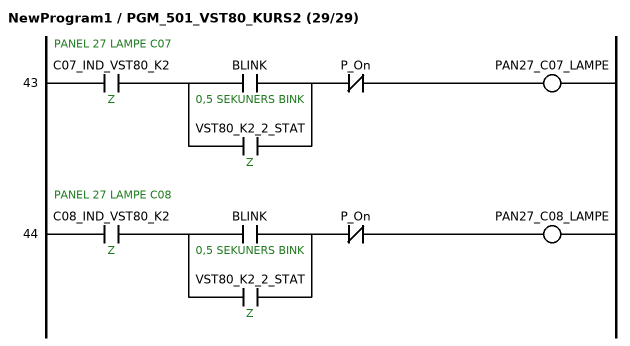
; [picture p528: NewProgram1 / PGM_501_VST80_KURS2, rungs 43-44]
; rung 43: PANEL 27 LAMPE C07
LD C07_IND_VST80_K2  ; Z
LD BLINK  ; 0,5 SEKUNERS BINK
OR VST80_K2_2_STAT  ; Z
ANDLD
ANDNOT P_On
OUT PAN27_C07_LAMPE
; rung 44: PANEL 27 LAMPE C08
LD C08_IND_VST80_K2  ; Z
LD BLINK  ; 0,5 SEKUNERS BINK
OR VST80_K2_2_STAT  ; Z
ANDLD
ANDNOT P_On
OUT PAN27_C08_LAMPE
; rung 45: Ingen_kommentar_funnet

### Section PGM_502_VST80_KURS3

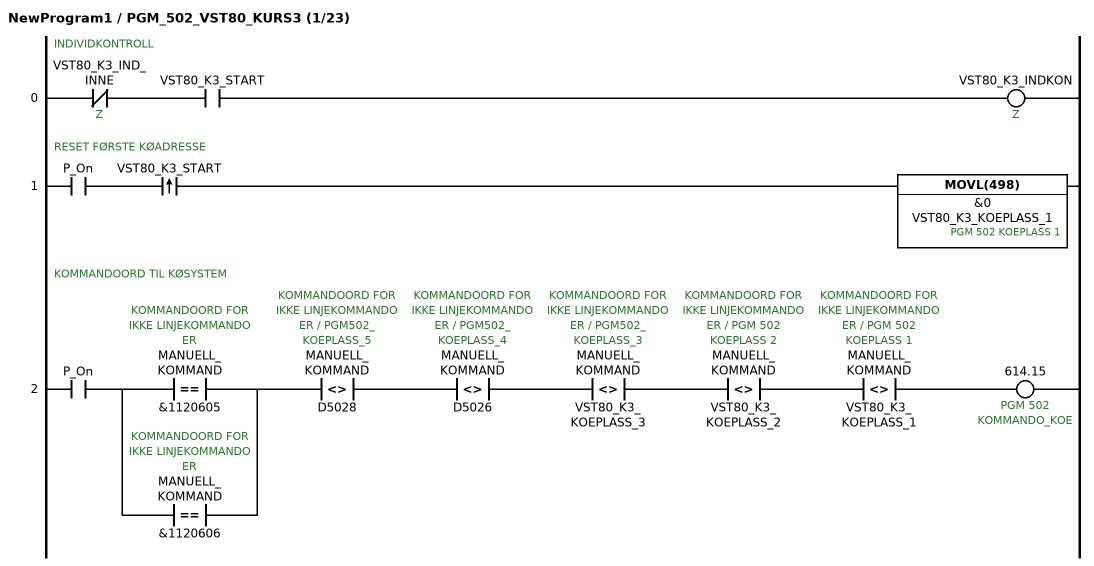
; rung 0: INDIVIDKONTROLL
LDNOT VST80_K3_IND_INNE  ; Z
AND VST80_K3_START
OUT VST80_K3_INDKON  ; Z
; rung 1: RESET FØRSTE KØADRESSE
LD P_On
@AND VST80_K3_START
MOVL(498) &0 VST80_K3_KOEPLASS_1  ; PGM 502 KOEPLASS 1
; rung 2: KOMMANDOORD TIL KØSYSTEM
LD P_On
LD=L(301) MANUELL_KOMMAND &1120605  ; KOMMANDOORD FOR IKKE LINJEKOMMANDOER
OR=L(301) MANUELL_KOMMAND &1120606  ; KOMMANDOORD FOR IKKE LINJEKOMMANDOER
ANDLD
AND<>L(306) MANUELL_KOMMAND D5028  ; KOMMANDOORD FOR IKKE LINJEKOMMANDOER, PGM502_KOEPLASS_5
AND<>L(306) MANUELL_KOMMAND D5026  ; KOMMANDOORD FOR IKKE LINJEKOMMANDOER, PGM502_KOEPLASS_4
AND<>L(306) MANUELL_KOMMAND VST80_K3_KOEPLASS_3  ; KOMMANDOORD FOR IKKE LINJEKOMMANDOER, PGM502_KOEPLASS_3
AND<>L(306) MANUELL_KOMMAND VST80_K3_KOEPLASS_2  ; KOMMANDOORD FOR IKKE LINJEKOMMANDOER, PGM 502 KOEPLASS 2
AND<>L(306) MANUELL_KOMMAND VST80_K3_KOEPLASS_1  ; KOMMANDOORD FOR IKKE LINJEKOMMANDOER, PGM 502 KOEPLASS 1
OUT 614.15  ; PGM 502 KOMMANDO_KOE

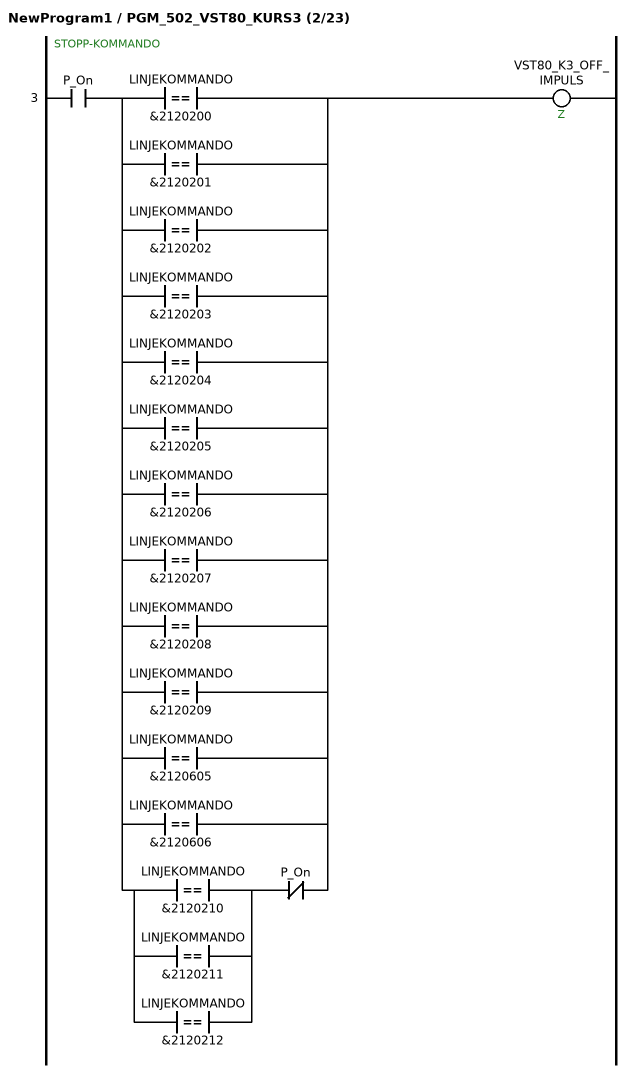
; rung 3: STOPP-KOMMANDO
LD P_On
LD=L(301) LINJEKOMMANDO &2120200
OR=L(301) LINJEKOMMANDO &2120201
OR=L(301) LINJEKOMMANDO &2120202
OR=L(301) LINJEKOMMANDO &2120203
OR=L(301) LINJEKOMMANDO &2120204
OR=L(301) LINJEKOMMANDO &2120205
OR=L(301) LINJEKOMMANDO &2120206
OR=L(301) LINJEKOMMANDO &2120207
OR=L(301) LINJEKOMMANDO &2120208
OR=L(301) LINJEKOMMANDO &2120209
OR=L(301) LINJEKOMMANDO &2120605
OR=L(301) LINJEKOMMANDO &2120606
LD=L(301) LINJEKOMMANDO &2120210
OR=L(301) LINJEKOMMANDO &2120211
OR=L(301) LINJEKOMMANDO &2120212
ANDNOT P_On
ORLD
ANDLD
OUT VST80_K3_OFF_IMPULS  ; Z

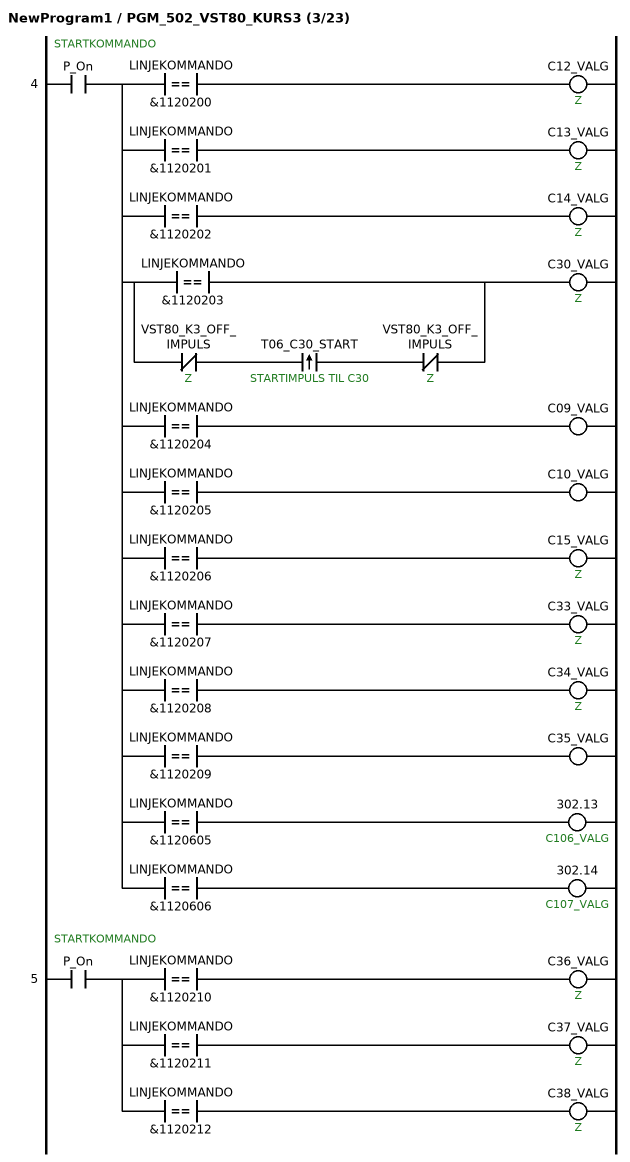
; rung 4: STARTKOMMANDO
LD P_On
OUT TR0
AND=L(301) LINJEKOMMANDO &1120200
OUT C12_VALG  ; Z
LD TR0
AND=L(301) LINJEKOMMANDO &1120201
OUT C13_VALG  ; Z
LD TR0
AND=L(301) LINJEKOMMANDO &1120202
OUT C14_VALG  ; Z
LD TR0
LD=L(301) LINJEKOMMANDO &1120203
LDNOT VST80_K3_OFF_IMPULS  ; Z
@AND T06_C30_START  ; STARTIMPULS TIL C30
ANDNOT VST80_K3_OFF_IMPULS  ; Z
ORLD
ANDLD
OUT C30_VALG  ; Z
LD TR0
AND=L(301) LINJEKOMMANDO &1120204
OUT C09_VALG
LD TR0
AND=L(301) LINJEKOMMANDO &1120205
OUT C10_VALG
LD TR0
AND=L(301) LINJEKOMMANDO &1120206
OUT C15_VALG  ; Z
LD TR0
AND=L(301) LINJEKOMMANDO &1120207
OUT C33_VALG  ; Z
LD TR0
AND=L(301) LINJEKOMMANDO &1120208
OUT C34_VALG  ; Z
LD TR0
AND=L(301) LINJEKOMMANDO &1120209
OUT C35_VALG
LD TR0
AND=L(301) LINJEKOMMANDO &1120605
OUT 302.13  ; C106_VALG
LD TR0
AND=L(301) LINJEKOMMANDO &1120606
OUT 302.14  ; C107_VALG
; rung 5: STARTKOMMANDO
LD P_On
OUT TR0
AND=L(301) LINJEKOMMANDO &1120210
OUT C36_VALG  ; Z
LD TR0
AND=L(301) LINJEKOMMANDO &1120211
OUT C37_VALG  ; Z
LD TR0
AND=L(301) LINJEKOMMANDO &1120212
OUT C38_VALG  ; Z

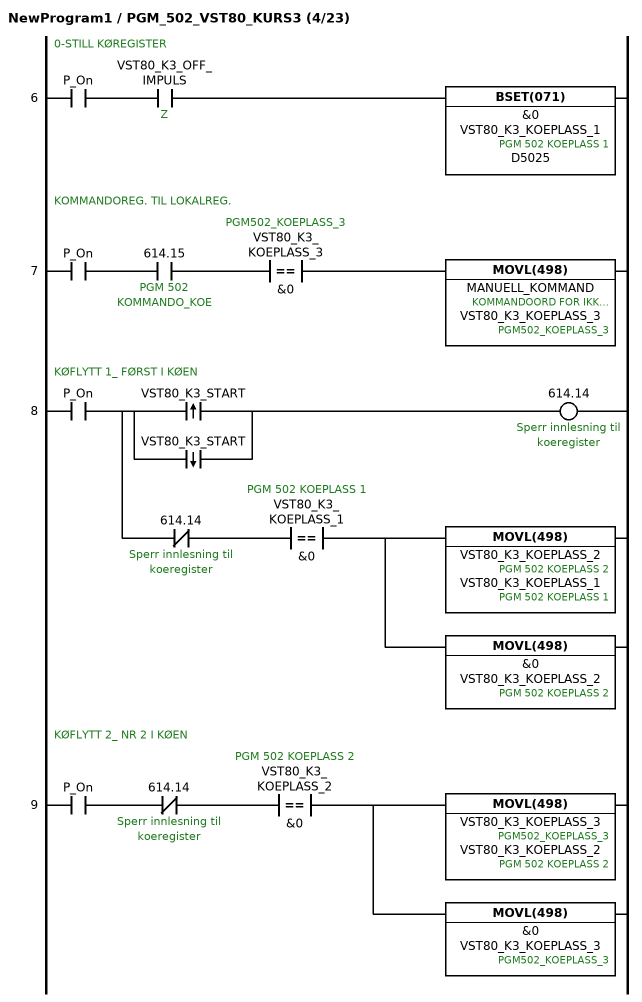
; rung 6: 0-STILL KØREGISTER
LD P_On
AND VST80_K3_OFF_IMPULS  ; Z
BSET(071) &0 VST80_K3_KOEPLASS_1 D5025  ; PGM 502 KOEPLASS 1
; rung 7: KOMMANDOREG. TIL LOKALREG.
LD P_On
AND 614.15  ; PGM 502 KOMMANDO_KOE
AND=L(301) VST80_K3_KOEPLASS_3 &0  ; PGM502_KOEPLASS_3
MOVL(498) MANUELL_KOMMAND VST80_K3_KOEPLASS_3  ; KOMMANDOORD FOR IKKE LINJEKOMMANDOER, PGM502_KOEPLASS_3
; rung 8: KØFLYTT 1_ FØRST I KØEN
LD P_On
OUT TR0
@LD VST80_K3_START
%OR VST80_K3_START
ANDLD
OUT 614.14  ; Sperr innlesning til koeregister
LD TR0
ANDNOT 614.14  ; Sperr innlesning til koeregister
AND=L(301) VST80_K3_KOEPLASS_1 &0  ; PGM 502 KOEPLASS 1
MOVL(498) VST80_K3_KOEPLASS_2 VST80_K3_KOEPLASS_1  ; PGM 502 KOEPLASS 2, PGM 502 KOEPLASS 1
MOVL(498) &0 VST80_K3_KOEPLASS_2  ; PGM 502 KOEPLASS 2
; rung 9: KØFLYTT 2_ NR 2 I KØEN
LD P_On
ANDNOT 614.14  ; Sperr innlesning til koeregister
AND=L(301) VST80_K3_KOEPLASS_2 &0  ; PGM 502 KOEPLASS 2
MOVL(498) VST80_K3_KOEPLASS_3 VST80_K3_KOEPLASS_2  ; PGM502_KOEPLASS_3, PGM 502 KOEPLASS 2
MOVL(498) &0 VST80_K3_KOEPLASS_3  ; PGM502_KOEPLASS_3

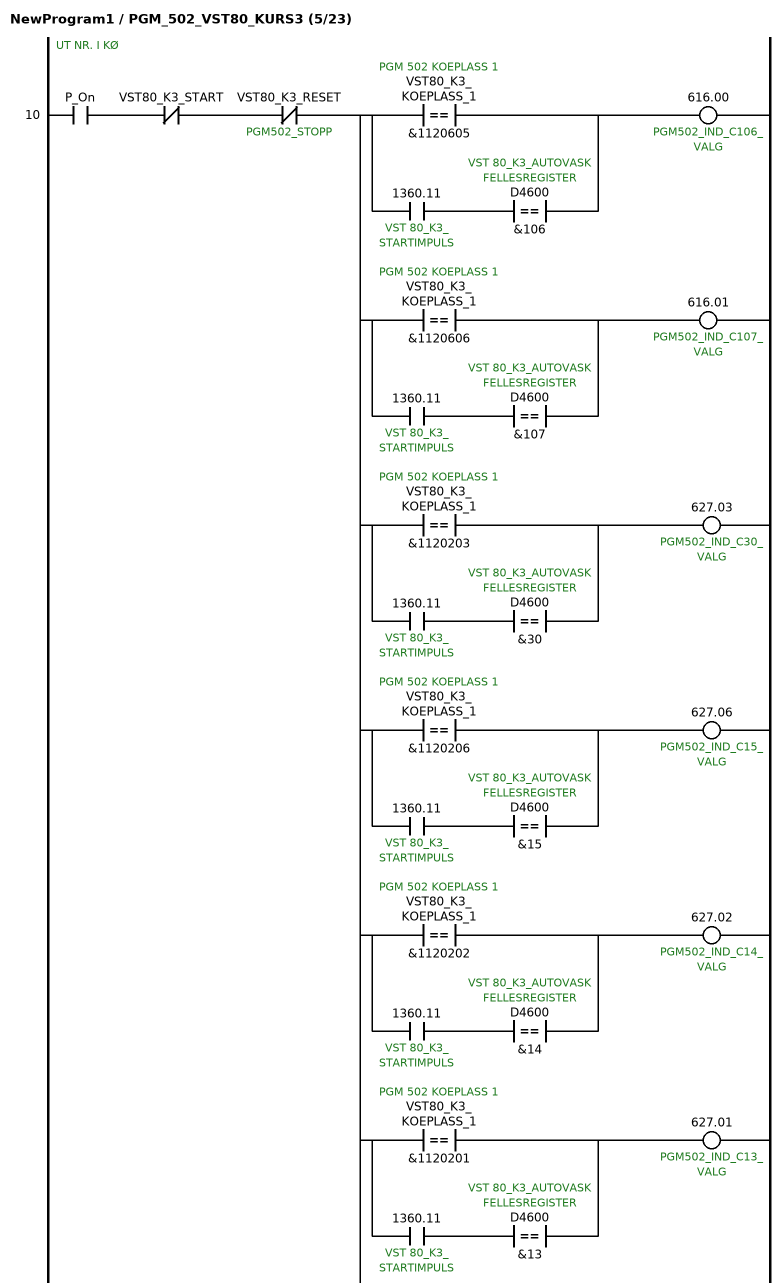

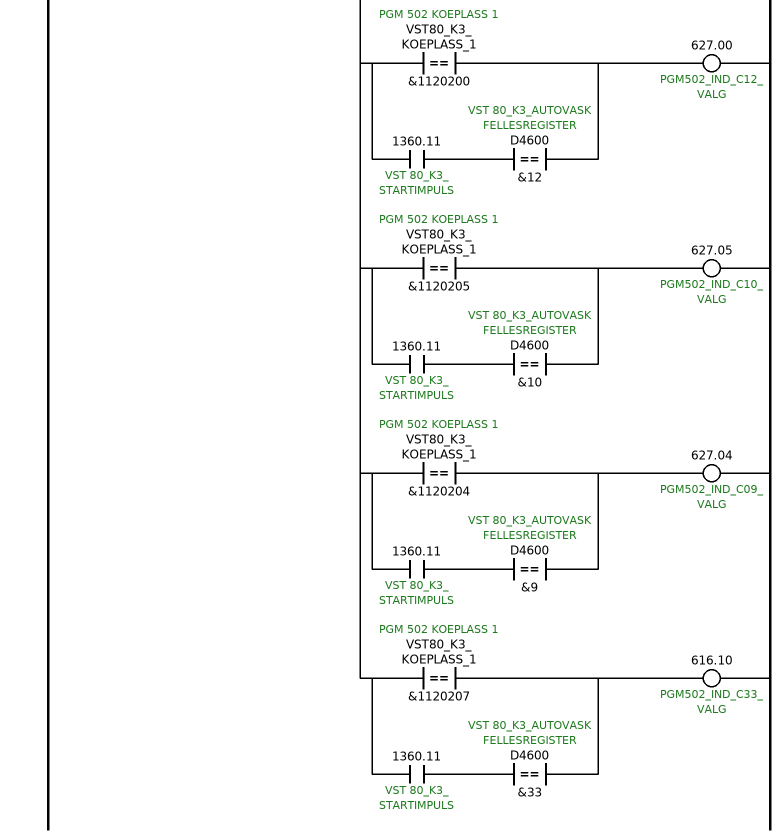
; rung 10: UT NR. I KØ
LD P_On
ANDNOT VST80_K3_START
ANDNOT VST80_K3_RESET  ; PGM502_STOPP
OUT TR0
LD=L(301) VST80_K3_KOEPLASS_1 &1120605  ; PGM 502 KOEPLASS 1
LD 1360.11  ; VST 80_K3_STARTIMPULS
AND=(300) D4600 &106  ; VST 80_K3_AUTOVASK FELLESREGISTER
ORLD
ANDLD
OUT 616.00  ; PGM502_IND_C106_VALG
LD TR0
LD=L(301) VST80_K3_KOEPLASS_1 &1120606  ; PGM 502 KOEPLASS 1
LD 1360.11  ; VST 80_K3_STARTIMPULS
AND=(300) D4600 &107  ; VST 80_K3_AUTOVASK FELLESREGISTER
ORLD
ANDLD
OUT 616.01  ; PGM502_IND_C107_VALG
LD TR0
LD=L(301) VST80_K3_KOEPLASS_1 &1120203  ; PGM 502 KOEPLASS 1
LD 1360.11  ; VST 80_K3_STARTIMPULS
AND=(300) D4600 &30  ; VST 80_K3_AUTOVASK FELLESREGISTER
ORLD
ANDLD
OUT 627.03  ; PGM502_IND_C30_VALG
LD TR0
LD=L(301) VST80_K3_KOEPLASS_1 &1120206  ; PGM 502 KOEPLASS 1
LD 1360.11  ; VST 80_K3_STARTIMPULS
AND=(300) D4600 &15  ; VST 80_K3_AUTOVASK FELLESREGISTER
ORLD
ANDLD
OUT 627.06  ; PGM502_IND_C15_VALG
LD TR0
LD=L(301) VST80_K3_KOEPLASS_1 &1120202  ; PGM 502 KOEPLASS 1
LD 1360.11  ; VST 80_K3_STARTIMPULS
AND=(300) D4600 &14  ; VST 80_K3_AUTOVASK FELLESREGISTER
ORLD
ANDLD
OUT 627.02  ; PGM502_IND_C14_VALG
LD TR0
LD=L(301) VST80_K3_KOEPLASS_1 &1120201  ; PGM 502 KOEPLASS 1
LD 1360.11  ; VST 80_K3_STARTIMPULS
AND=(300) D4600 &13  ; VST 80_K3_AUTOVASK FELLESREGISTER
ORLD
ANDLD
OUT 627.01  ; PGM502_IND_C13_VALG
LD TR0
LD=L(301) VST80_K3_KOEPLASS_1 &1120200  ; PGM 502 KOEPLASS 1
LD 1360.11  ; VST 80_K3_STARTIMPULS
AND=(300) D4600 &12  ; VST 80_K3_AUTOVASK FELLESREGISTER
ORLD
ANDLD
OUT 627.00  ; PGM502_IND_C12_VALG
LD TR0
LD=L(301) VST80_K3_KOEPLASS_1 &1120205  ; PGM 502 KOEPLASS 1
LD 1360.11  ; VST 80_K3_STARTIMPULS
AND=(300) D4600 &10  ; VST 80_K3_AUTOVASK FELLESREGISTER
ORLD
ANDLD
OUT 627.05  ; PGM502_IND_C10_VALG
LD TR0
LD=L(301) VST80_K3_KOEPLASS_1 &1120204  ; PGM 502 KOEPLASS 1
LD 1360.11  ; VST 80_K3_STARTIMPULS
AND=(300) D4600 &9  ; VST 80_K3_AUTOVASK FELLESREGISTER
ORLD
ANDLD
OUT 627.04  ; PGM502_IND_C09_VALG
LD TR0
LD=L(301) VST80_K3_KOEPLASS_1 &1120207  ; PGM 502 KOEPLASS 1
LD 1360.11  ; VST 80_K3_STARTIMPULS
AND=(300) D4600 &33  ; VST 80_K3_AUTOVASK FELLESREGISTER
ORLD
ANDLD
OUT 616.10  ; PGM502_IND_C33_VALG

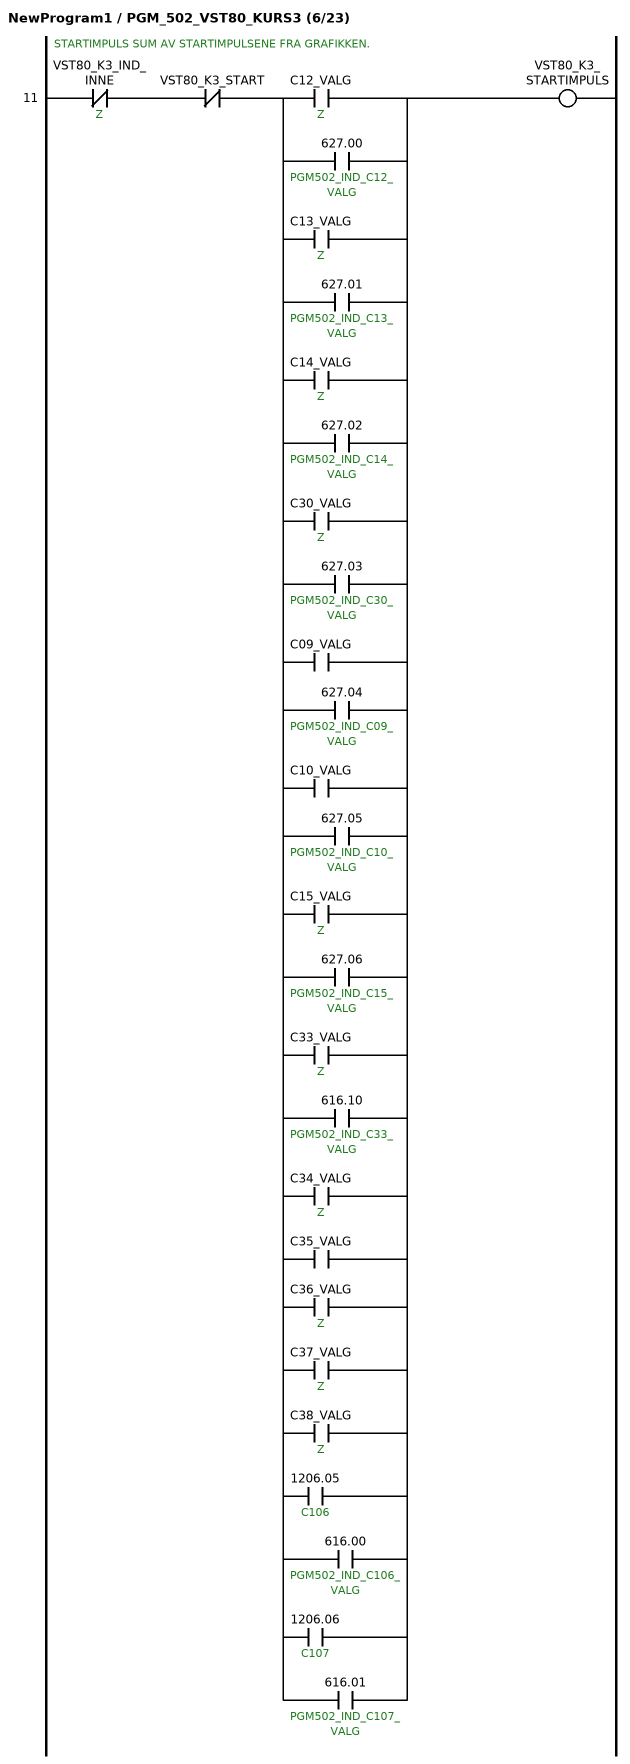
; rung 11: STARTIMPULS SUM AV STARTIMPULSENE FRA GRAFIKKEN.
LDNOT VST80_K3_IND_INNE  ; Z
ANDNOT VST80_K3_START
LD C12_VALG  ; Z
OR 627.00  ; PGM502_IND_C12_VALG
OR C13_VALG  ; Z
OR 627.01  ; PGM502_IND_C13_VALG
OR C14_VALG  ; Z
OR 627.02  ; PGM502_IND_C14_VALG
OR C30_VALG  ; Z
OR 627.03  ; PGM502_IND_C30_VALG
OR C09_VALG
OR 627.04  ; PGM502_IND_C09_VALG
OR C10_VALG
OR 627.05  ; PGM502_IND_C10_VALG
OR C15_VALG  ; Z
OR 627.06  ; PGM502_IND_C15_VALG
OR C33_VALG  ; Z
OR 616.10  ; PGM502_IND_C33_VALG
OR C34_VALG  ; Z
OR C35_VALG
OR C36_VALG  ; Z
OR C37_VALG  ; Z
OR C38_VALG  ; Z
OR 1206.05  ; C106
OR 616.00  ; PGM502_IND_C106_VALG
OR 1206.06  ; C107
OR 616.01  ; PGM502_IND_C107_VALG
ANDLD
OUT VST80_K3_STARTIMPULS

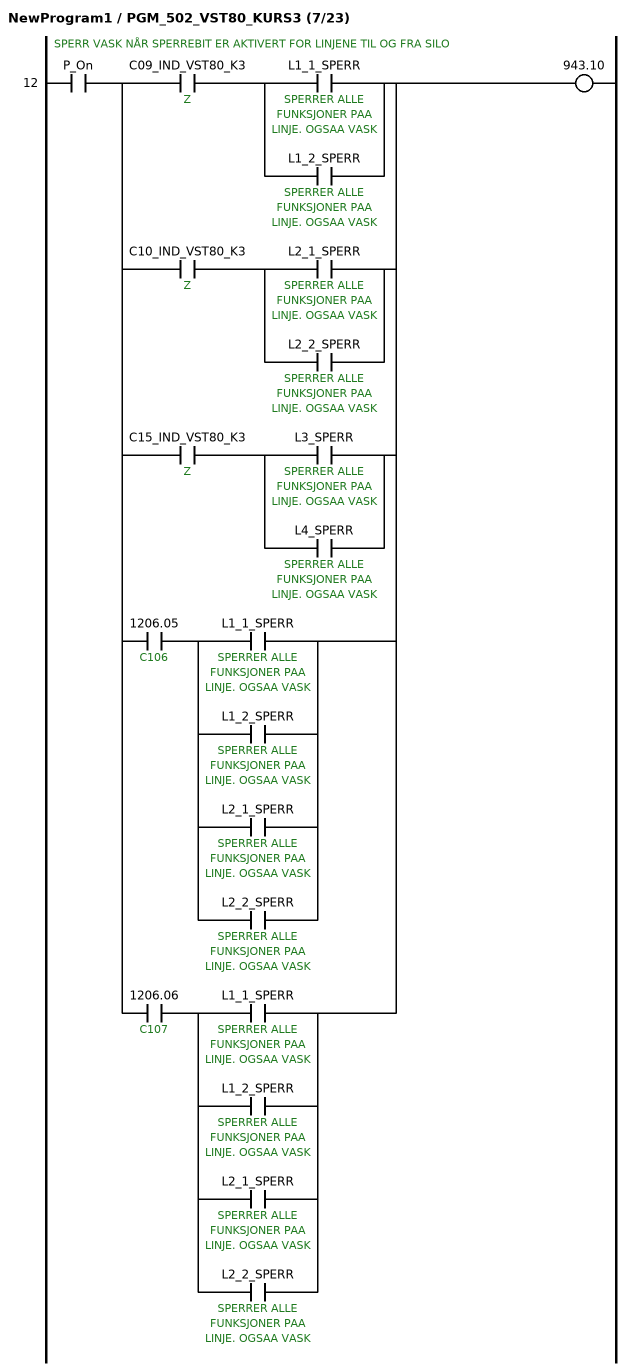
; rung 12: SPERR VASK NÅR SPERREBIT ER AKTIVERT FOR LINJENE TIL OG FRA SILO
LD P_On
LD C09_IND_VST80_K3  ; Z
LD L1_1_SPERR  ; SPERRER ALLE FUNKSJONER PAA LINJE. OGSAA VASK
OR L1_2_SPERR  ; SPERRER ALLE FUNKSJONER PAA LINJE. OGSAA VASK
ANDLD
LD C10_IND_VST80_K3  ; Z
LD L2_1_SPERR  ; SPERRER ALLE FUNKSJONER PAA LINJE. OGSAA VASK
OR L2_2_SPERR  ; SPERRER ALLE FUNKSJONER PAA LINJE. OGSAA VASK
ANDLD
ORLD
LD C15_IND_VST80_K3  ; Z
LD L3_SPERR  ; SPERRER ALLE FUNKSJONER PAA LINJE. OGSAA VASK
OR L4_SPERR  ; SPERRER ALLE FUNKSJONER PAA LINJE. OGSAA VASK
ANDLD
ORLD
LD 1206.05  ; C106
LD L1_1_SPERR  ; SPERRER ALLE FUNKSJONER PAA LINJE. OGSAA VASK
OR L1_2_SPERR  ; SPERRER ALLE FUNKSJONER PAA LINJE. OGSAA VASK
OR L2_1_SPERR  ; SPERRER ALLE FUNKSJONER PAA LINJE. OGSAA VASK
OR L2_2_SPERR  ; SPERRER ALLE FUNKSJONER PAA LINJE. OGSAA VASK
ANDLD
ORLD
LD 1206.06  ; C107
LD L1_1_SPERR  ; SPERRER ALLE FUNKSJONER PAA LINJE. OGSAA VASK
OR L1_2_SPERR  ; SPERRER ALLE FUNKSJONER PAA LINJE. OGSAA VASK
OR L2_1_SPERR  ; SPERRER ALLE FUNKSJONER PAA LINJE. OGSAA VASK
OR L2_2_SPERR  ; SPERRER ALLE FUNKSJONER PAA LINJE. OGSAA VASK
ANDLD
ORLD
ANDLD
OUT 943.10

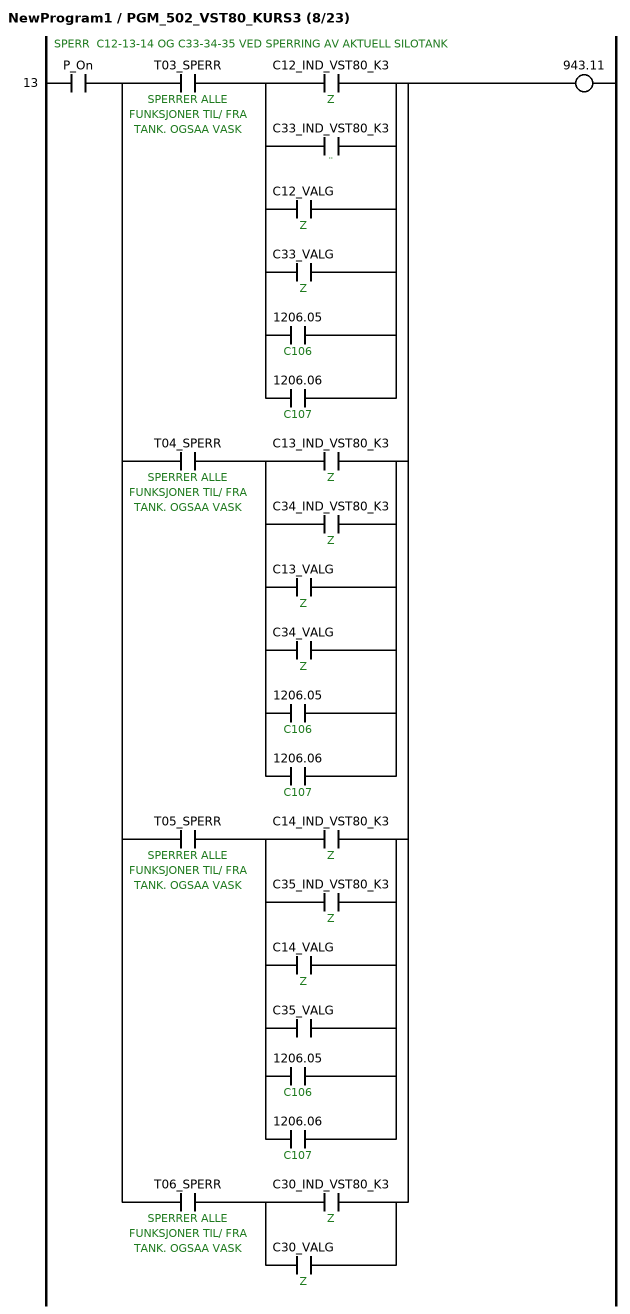
; rung 13: SPERR  C12-13-14 OG C33-34-35 VED SPERRING AV AKTUELL SILOTANK
LD P_On
LD T03_SPERR  ; SPERRER ALLE FUNKSJONER TIL/ FRA TANK. OGSAA VASK
LD C12_IND_VST80_K3  ; Z
OR C33_IND_VST80_K3  ; ¨
OR C12_VALG  ; Z
OR C33_VALG  ; Z
OR 1206.05  ; C106
OR 1206.06  ; C107
ANDLD
LD T04_SPERR  ; SPERRER ALLE FUNKSJONER TIL/ FRA TANK. OGSAA VASK
LD C13_IND_VST80_K3  ; Z
OR C34_IND_VST80_K3  ; Z
OR C13_VALG  ; Z
OR C34_VALG  ; Z
OR 1206.05  ; C106
OR 1206.06  ; C107
ANDLD
ORLD
LD T05_SPERR  ; SPERRER ALLE FUNKSJONER TIL/ FRA TANK. OGSAA VASK
LD C14_IND_VST80_K3  ; Z
OR C35_IND_VST80_K3  ; Z
OR C14_VALG  ; Z
OR C35_VALG
OR 1206.05  ; C106
OR 1206.06  ; C107
ANDLD
ORLD
LD T06_SPERR  ; SPERRER ALLE FUNKSJONER TIL/ FRA TANK. OGSAA VASK
LD C30_IND_VST80_K3  ; Z
OR C30_VALG  ; Z
ANDLD
ORLD
ANDLD
OUT 943.11

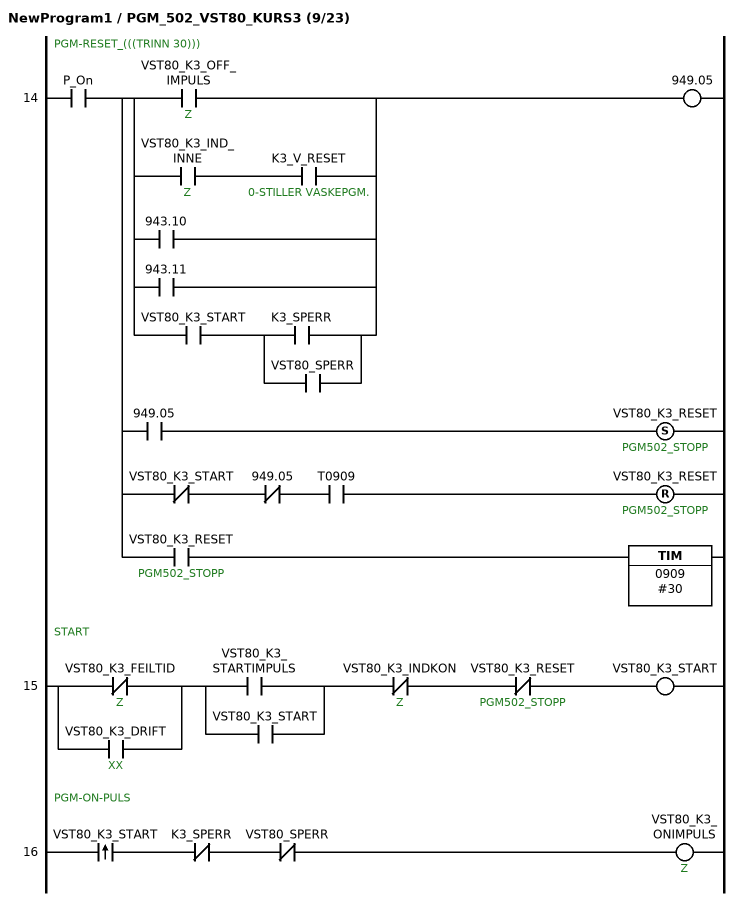
; rung 14: PGM-RESET_(((TRINN 30)))
LD P_On
OUT TR0
LD VST80_K3_OFF_IMPULS  ; Z
LD VST80_K3_IND_INNE  ; Z
AND K3_V_RESET  ; 0-STILLER VASKEPGM.
ORLD
OR 943.10
OR 943.11
LD VST80_K3_START
LD K3_SPERR
OR VST80_SPERR
ANDLD
ORLD
ANDLD
OUT 949.05
LD TR0
AND 949.05
SET VST80_K3_RESET  ; PGM502_STOPP
LD TR0
ANDNOT VST80_K3_START
ANDNOT 949.05
AND T0909
RSET VST80_K3_RESET  ; PGM502_STOPP
LD TR0
AND VST80_K3_RESET  ; PGM502_STOPP
TIM 0909 #30
; rung 15: START
LDNOT VST80_K3_FEILTID  ; Z
OR VST80_K3_DRIFT  ; XX
LD VST80_K3_STARTIMPULS
OR VST80_K3_START
ANDLD
ANDNOT VST80_K3_INDKON  ; Z
ANDNOT VST80_K3_RESET  ; PGM502_STOPP
OUT VST80_K3_START
; rung 16: PGM-ON-PULS
@LD VST80_K3_START
ANDNOT K3_SPERR
ANDNOT VST80_SPERR
OUT VST80_K3_ONIMPULS  ; Z

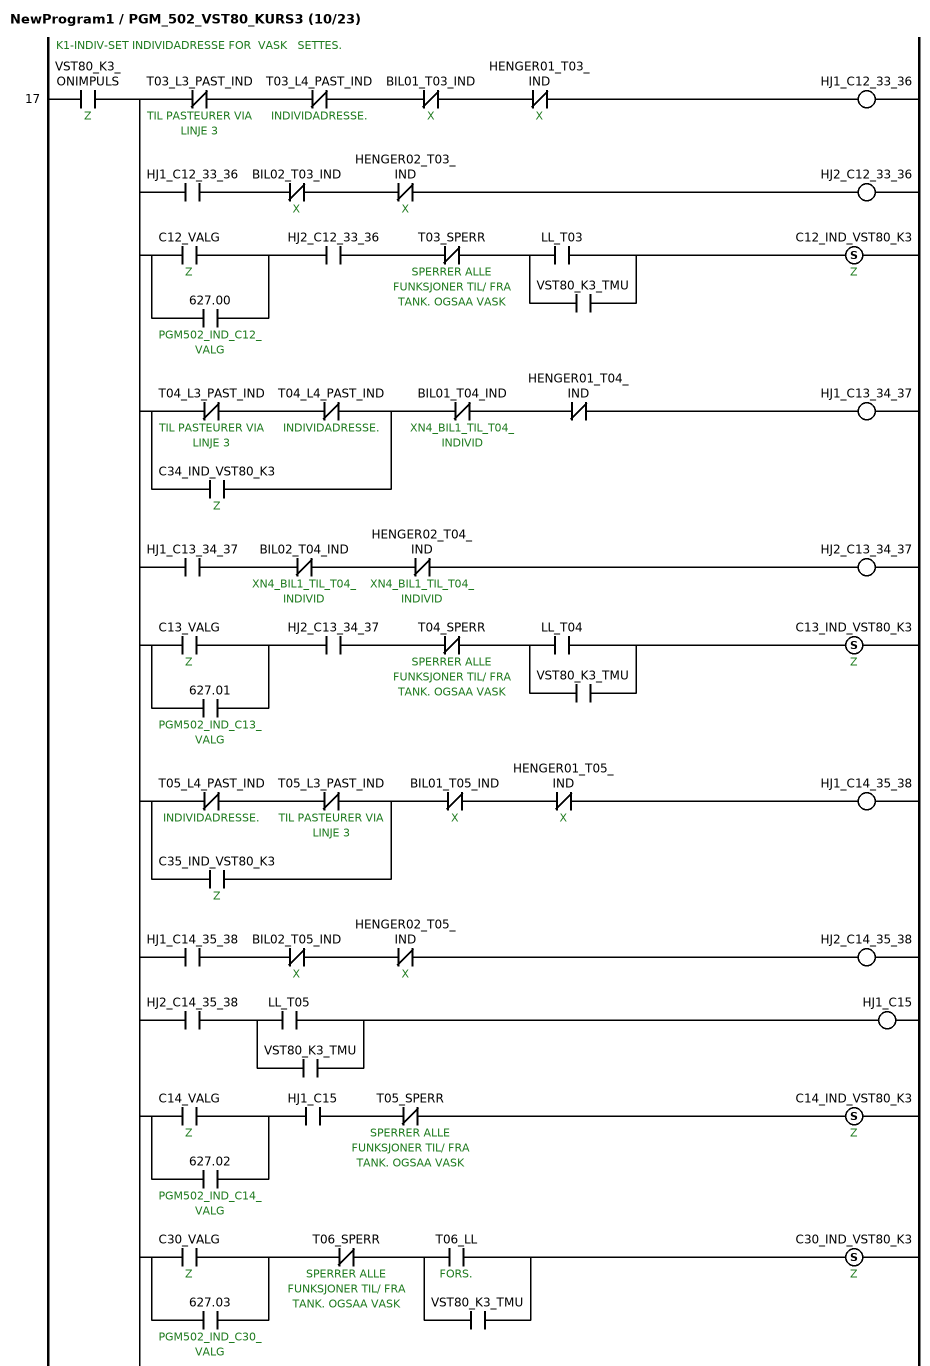

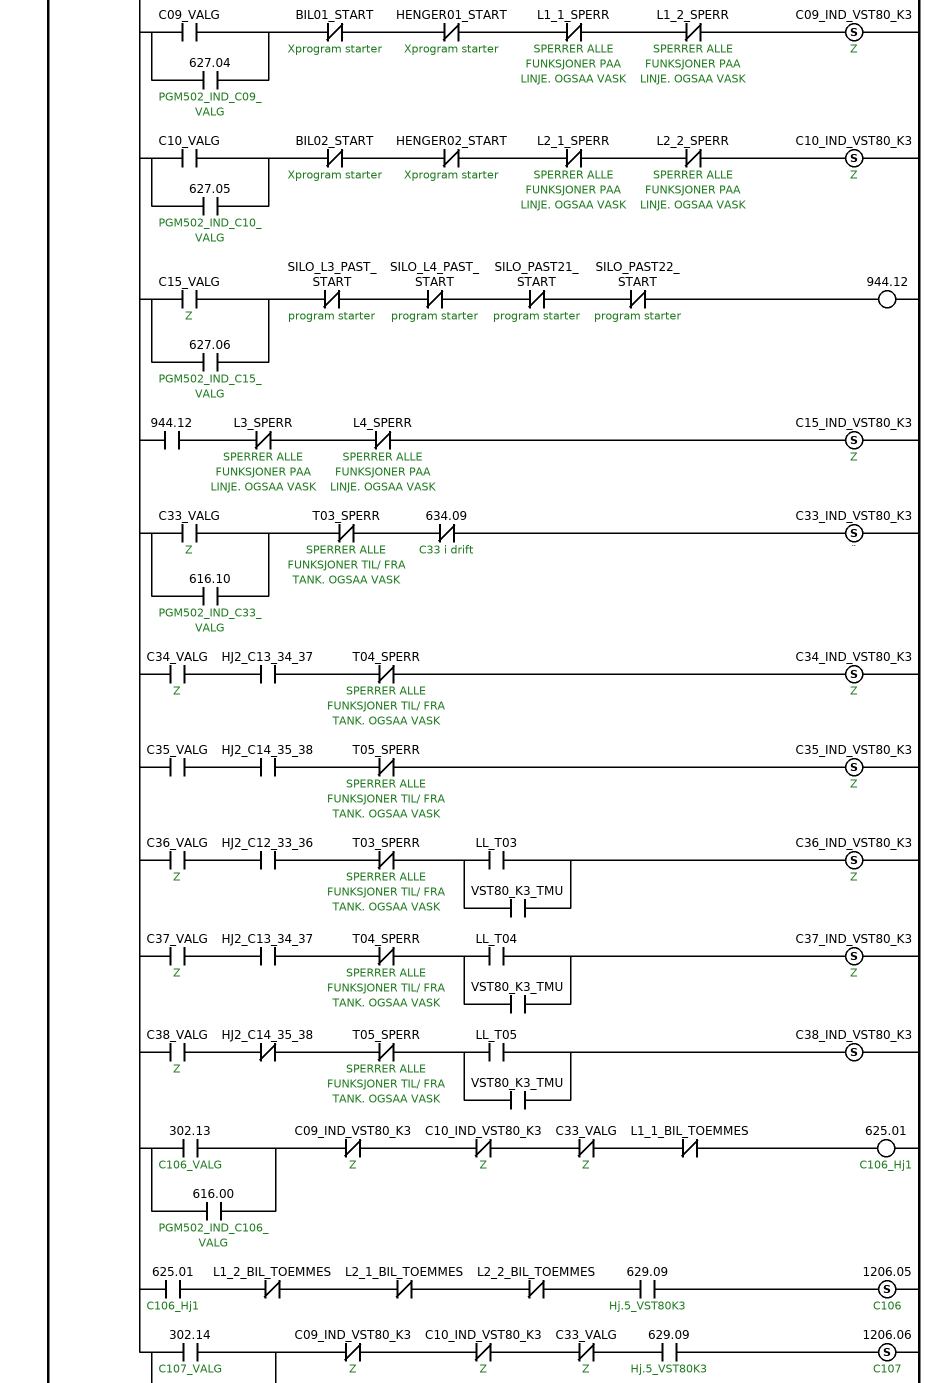

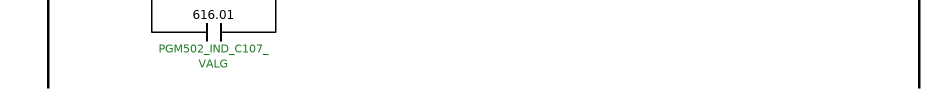
; rung 17: K1-INDIV-SET INDIVIDADRESSE FOR  VASK   SETTES.
LD VST80_K3_ONIMPULS  ; Z
OUT TR0
ANDNOT T03_L3_PAST_IND  ; TIL PASTEURER VIA LINJE 3
ANDNOT T03_L4_PAST_IND  ; INDIVIDADRESSE.
ANDNOT BIL01_T03_IND  ; X
ANDNOT HENGER01_T03_IND  ; X
OUT HJ1_C12_33_36
LD TR0
AND HJ1_C12_33_36
ANDNOT BIL02_T03_IND  ; X
ANDNOT HENGER02_T03_IND  ; X
OUT HJ2_C12_33_36
LD TR0
LD C12_VALG  ; Z
OR 627.00  ; PGM502_IND_C12_VALG
ANDLD
AND HJ2_C12_33_36
ANDNOT T03_SPERR  ; SPERRER ALLE FUNKSJONER TIL/ FRA TANK. OGSAA VASK
LD LL_T03
OR VST80_K3_TMU
ANDLD
SET C12_IND_VST80_K3  ; Z
LD TR0
LDNOT T04_L3_PAST_IND  ; TIL PASTEURER VIA LINJE 3
ANDNOT T04_L4_PAST_IND  ; INDIVIDADRESSE.
OR C34_IND_VST80_K3  ; Z
ANDLD
ANDNOT BIL01_T04_IND  ; XN4_BIL1_TIL_T04_INDIVID
ANDNOT HENGER01_T04_IND
OUT HJ1_C13_34_37
LD TR0
AND HJ1_C13_34_37
ANDNOT BIL02_T04_IND  ; XN4_BIL1_TIL_T04_INDIVID
ANDNOT HENGER02_T04_IND  ; XN4_BIL1_TIL_T04_INDIVID
OUT HJ2_C13_34_37
LD TR0
LD C13_VALG  ; Z
OR 627.01  ; PGM502_IND_C13_VALG
ANDLD
AND HJ2_C13_34_37
ANDNOT T04_SPERR  ; SPERRER ALLE FUNKSJONER TIL/ FRA TANK. OGSAA VASK
LD LL_T04
OR VST80_K3_TMU
ANDLD
SET C13_IND_VST80_K3  ; Z
LD TR0
LDNOT T05_L4_PAST_IND  ; INDIVIDADRESSE.
ANDNOT T05_L3_PAST_IND  ; TIL PASTEURER VIA LINJE 3
OR C35_IND_VST80_K3  ; Z
ANDLD
ANDNOT BIL01_T05_IND  ; X
ANDNOT HENGER01_T05_IND  ; X
OUT HJ1_C14_35_38
LD TR0
AND HJ1_C14_35_38
ANDNOT BIL02_T05_IND  ; X
ANDNOT HENGER02_T05_IND  ; X
OUT HJ2_C14_35_38
LD TR0
AND HJ2_C14_35_38
LD LL_T05
OR VST80_K3_TMU
ANDLD
OUT HJ1_C15
LD TR0
LD C14_VALG  ; Z
OR 627.02  ; PGM502_IND_C14_VALG
ANDLD
AND HJ1_C15
ANDNOT T05_SPERR  ; SPERRER ALLE FUNKSJONER TIL/ FRA TANK. OGSAA VASK
SET C14_IND_VST80_K3  ; Z
LD TR0
LD C30_VALG  ; Z
OR 627.03  ; PGM502_IND_C30_VALG
ANDLD
ANDNOT T06_SPERR  ; SPERRER ALLE FUNKSJONER TIL/ FRA TANK. OGSAA VASK
LD T06_LL  ; FORS.
OR VST80_K3_TMU
ANDLD
SET C30_IND_VST80_K3  ; Z
LD TR0
LD C09_VALG
OR 627.04  ; PGM502_IND_C09_VALG
ANDLD
ANDNOT BIL01_START  ; Xprogram starter
ANDNOT HENGER01_START  ; Xprogram starter
ANDNOT L1_1_SPERR  ; SPERRER ALLE FUNKSJONER PAA LINJE. OGSAA VASK
ANDNOT L1_2_SPERR  ; SPERRER ALLE FUNKSJONER PAA LINJE. OGSAA VASK
SET C09_IND_VST80_K3  ; Z
LD TR0
LD C10_VALG
OR 627.05  ; PGM502_IND_C10_VALG
ANDLD
ANDNOT BIL02_START  ; Xprogram starter
ANDNOT HENGER02_START  ; Xprogram starter
ANDNOT L2_1_SPERR  ; SPERRER ALLE FUNKSJONER PAA LINJE. OGSAA VASK
ANDNOT L2_2_SPERR  ; SPERRER ALLE FUNKSJONER PAA LINJE. OGSAA VASK
SET C10_IND_VST80_K3  ; Z
LD TR0
LD C15_VALG  ; Z
OR 627.06  ; PGM502_IND_C15_VALG
ANDLD
ANDNOT SILO_L3_PAST_START  ; program starter
ANDNOT SILO_L4_PAST_START  ; program starter
ANDNOT SILO_PAST21_START  ; program starter
ANDNOT SILO_PAST22_START  ; program starter
OUT 944.12
LD TR0
AND 944.12
ANDNOT L3_SPERR  ; SPERRER ALLE FUNKSJONER PAA LINJE. OGSAA VASK
ANDNOT L4_SPERR  ; SPERRER ALLE FUNKSJONER PAA LINJE. OGSAA VASK
SET C15_IND_VST80_K3  ; Z
LD TR0
LD C33_VALG  ; Z
OR 616.10  ; PGM502_IND_C33_VALG
ANDLD
ANDNOT T03_SPERR  ; SPERRER ALLE FUNKSJONER TIL/ FRA TANK. OGSAA VASK
ANDNOT 634.09  ; C33 i drift
SET C33_IND_VST80_K3  ; ¨
LD TR0
AND C34_VALG  ; Z
AND HJ2_C13_34_37
ANDNOT T04_SPERR  ; SPERRER ALLE FUNKSJONER TIL/ FRA TANK. OGSAA VASK
SET C34_IND_VST80_K3  ; Z
LD TR0
AND C35_VALG
AND HJ2_C14_35_38
ANDNOT T05_SPERR  ; SPERRER ALLE FUNKSJONER TIL/ FRA TANK. OGSAA VASK
SET C35_IND_VST80_K3  ; Z
LD TR0
AND C36_VALG  ; Z
AND HJ2_C12_33_36
ANDNOT T03_SPERR  ; SPERRER ALLE FUNKSJONER TIL/ FRA TANK. OGSAA VASK
LD LL_T03
OR VST80_K3_TMU
ANDLD
SET C36_IND_VST80_K3  ; Z
LD TR0
AND C37_VALG  ; Z
AND HJ2_C13_34_37
ANDNOT T04_SPERR  ; SPERRER ALLE FUNKSJONER TIL/ FRA TANK. OGSAA VASK
LD LL_T04
OR VST80_K3_TMU
ANDLD
SET C37_IND_VST80_K3  ; Z
LD TR0
AND C38_VALG  ; Z
ANDNOT HJ2_C14_35_38
ANDNOT T05_SPERR  ; SPERRER ALLE FUNKSJONER TIL/ FRA TANK. OGSAA VASK
LD LL_T05
OR VST80_K3_TMU
ANDLD
SET C38_IND_VST80_K3
LD TR0
LD 302.13  ; C106_VALG
OR 616.00  ; PGM502_IND_C106_VALG
ANDLD
ANDNOT C09_IND_VST80_K3  ; Z
ANDNOT C10_IND_VST80_K3  ; Z
ANDNOT C33_VALG  ; Z
ANDNOT L1_1_BIL_TOEMMES
OUT 625.01  ; C106_Hj1
LD TR0
AND 625.01  ; C106_Hj1
ANDNOT L1_2_BIL_TOEMMES
ANDNOT L2_1_BIL_TOEMMES
ANDNOT L2_2_BIL_TOEMMES
AND 629.09  ; Hj.5_VST80K3
SET 1206.05  ; C106
LD TR0
LD 302.14  ; C107_VALG
OR 616.01  ; PGM502_IND_C107_VALG
ANDLD
ANDNOT C09_IND_VST80_K3  ; Z
ANDNOT C10_IND_VST80_K3  ; Z
ANDNOT C33_VALG  ; Z
AND 629.09  ; Hj.5_VST80K3
SET 1206.06  ; C107

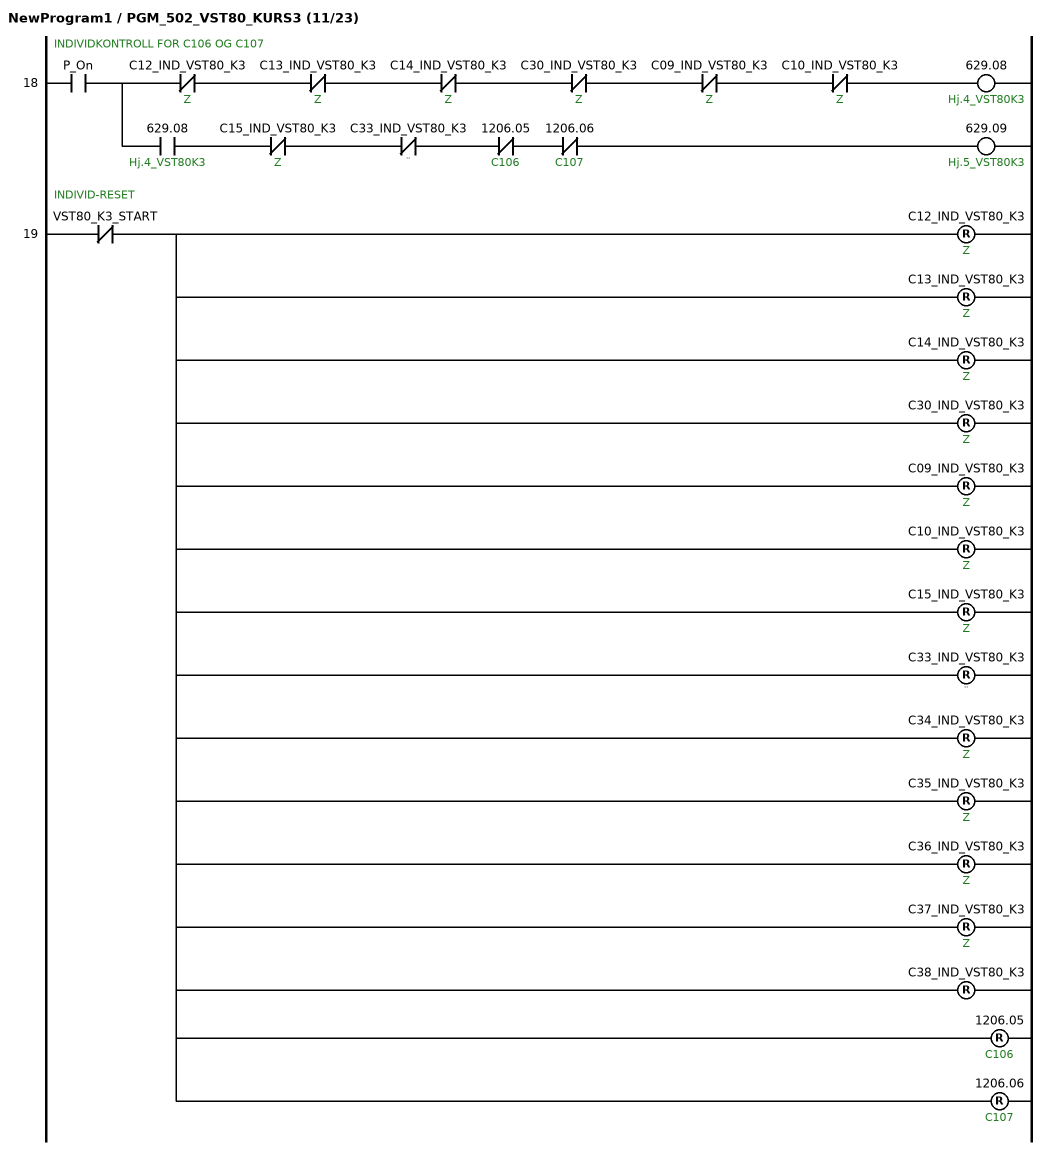
; rung 18: INDIVIDKONTROLL FOR C106 OG C107
LD P_On
OUT TR0
ANDNOT C12_IND_VST80_K3  ; Z
ANDNOT C13_IND_VST80_K3  ; Z
ANDNOT C14_IND_VST80_K3  ; Z
ANDNOT C30_IND_VST80_K3  ; Z
ANDNOT C09_IND_VST80_K3  ; Z
ANDNOT C10_IND_VST80_K3  ; Z
OUT 629.08  ; Hj.4_VST80K3
LD TR0
AND 629.08  ; Hj.4_VST80K3
ANDNOT C15_IND_VST80_K3  ; Z
ANDNOT C33_IND_VST80_K3  ; ¨
ANDNOT 1206.05  ; C106
ANDNOT 1206.06  ; C107
OUT 629.09  ; Hj.5_VST80K3
; rung 19: INDIVID-RESET
LDNOT VST80_K3_START
RSET C12_IND_VST80_K3  ; Z
RSET C13_IND_VST80_K3  ; Z
RSET C14_IND_VST80_K3  ; Z
RSET C30_IND_VST80_K3  ; Z
RSET C09_IND_VST80_K3  ; Z
RSET C10_IND_VST80_K3  ; Z
RSET C15_IND_VST80_K3  ; Z
RSET C33_IND_VST80_K3  ; ¨
RSET C34_IND_VST80_K3  ; Z
RSET C35_IND_VST80_K3  ; Z
RSET C36_IND_VST80_K3  ; Z
RSET C37_IND_VST80_K3  ; Z
RSET C38_IND_VST80_K3
RSET 1206.05  ; C106
RSET 1206.06  ; C107

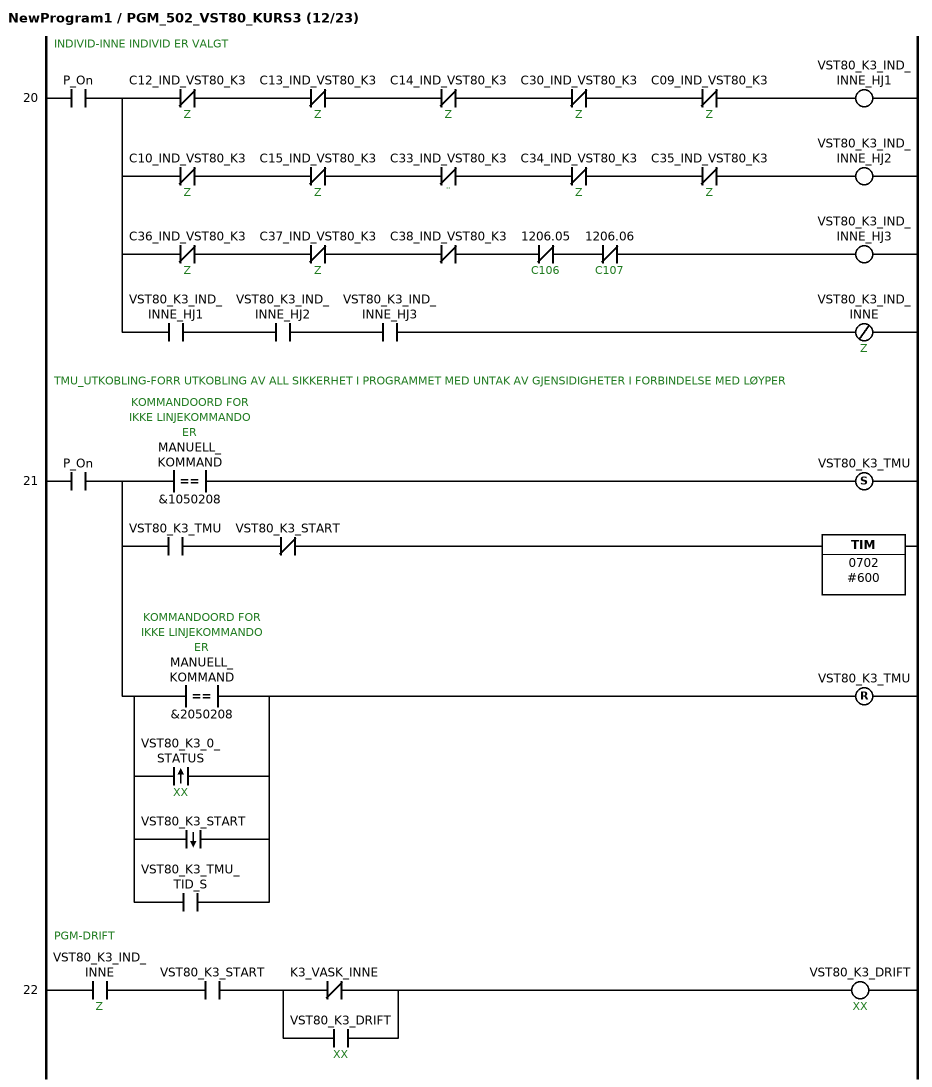
; rung 20: INDIVID-INNE INDIVID ER VALGT
LD P_On
OUT TR0
ANDNOT C12_IND_VST80_K3  ; Z
ANDNOT C13_IND_VST80_K3  ; Z
ANDNOT C14_IND_VST80_K3  ; Z
ANDNOT C30_IND_VST80_K3  ; Z
ANDNOT C09_IND_VST80_K3  ; Z
OUT VST80_K3_IND_INNE_HJ1
LD TR0
ANDNOT C10_IND_VST80_K3  ; Z
ANDNOT C15_IND_VST80_K3  ; Z
ANDNOT C33_IND_VST80_K3  ; ¨
ANDNOT C34_IND_VST80_K3  ; Z
ANDNOT C35_IND_VST80_K3  ; Z
OUT VST80_K3_IND_INNE_HJ2
LD TR0
ANDNOT C36_IND_VST80_K3  ; Z
ANDNOT C37_IND_VST80_K3  ; Z
ANDNOT C38_IND_VST80_K3
ANDNOT 1206.05  ; C106
ANDNOT 1206.06  ; C107
OUT VST80_K3_IND_INNE_HJ3
LD TR0
AND VST80_K3_IND_INNE_HJ1
AND VST80_K3_IND_INNE_HJ2
AND VST80_K3_IND_INNE_HJ3
OUTNOT VST80_K3_IND_INNE  ; Z
; rung 21: TMU_UTKOBLING-FORR UTKOBLING AV ALL SIKKERHET I PROGRAMMET MED UNTAK AV GJENSIDIGHETER I FORBINDELSE MED LØYPER
LD P_On
OUT TR0
AND=L(301) MANUELL_KOMMAND &1050208  ; KOMMANDOORD FOR IKKE LINJEKOMMANDOER
SET VST80_K3_TMU
LD TR0
AND VST80_K3_TMU
ANDNOT VST80_K3_START
TIM 0702 #600
LD TR0
LD=L(301) MANUELL_KOMMAND &2050208  ; KOMMANDOORD FOR IKKE LINJEKOMMANDOER
@OR VST80_K3_0_STATUS  ; XX
%OR VST80_K3_START
OR VST80_K3_TMU_TID_S
ANDLD
RSET VST80_K3_TMU
; rung 22: PGM-DRIFT
LD VST80_K3_IND_INNE  ; Z
AND VST80_K3_START
LDNOT K3_VASK_INNE
OR VST80_K3_DRIFT  ; XX
ANDLD
OUT VST80_K3_DRIFT  ; XX

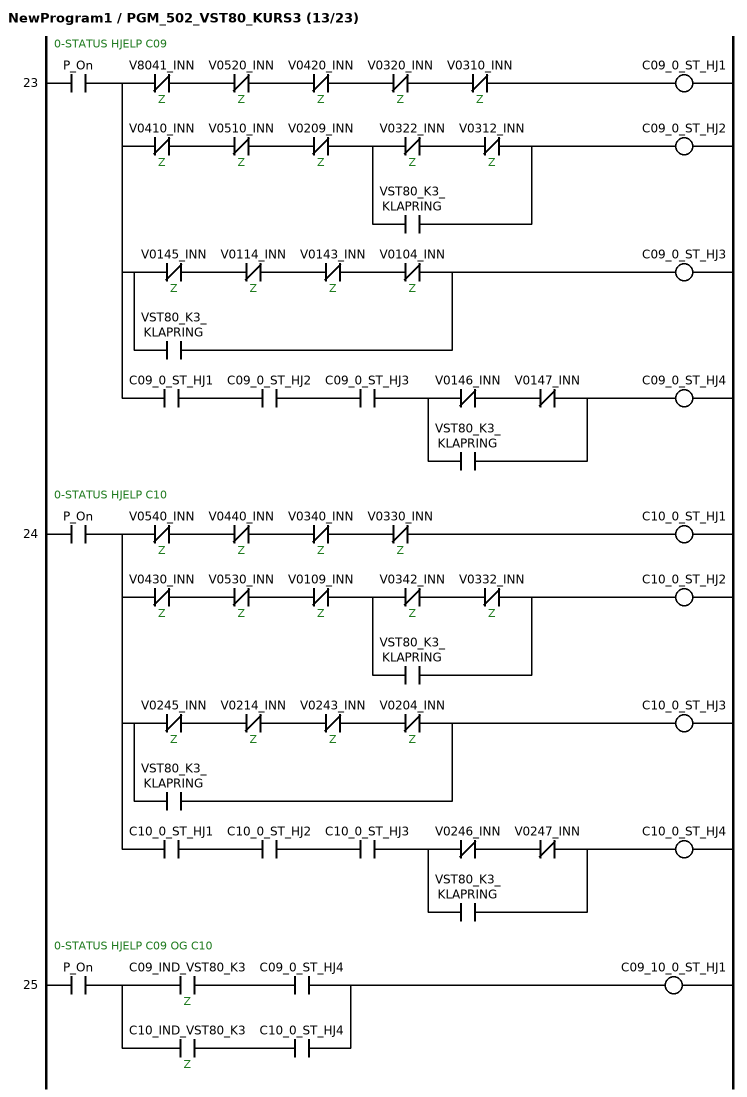
; rung 23: 0-STATUS HJELP C09
LD P_On
OUT TR0
ANDNOT V8041_INN  ; Z
ANDNOT V0520_INN  ; Z
ANDNOT V0420_INN  ; Z
ANDNOT V0320_INN  ; Z
ANDNOT V0310_INN  ; Z
OUT C09_0_ST_HJ1
LD TR0
ANDNOT V0410_INN  ; Z
ANDNOT V0510_INN  ; Z
ANDNOT V0209_INN  ; Z
LDNOT V0322_INN  ; Z
ANDNOT V0312_INN  ; Z
OR VST80_K3_KLAPRING
ANDLD
OUT C09_0_ST_HJ2
LD TR0
LDNOT V0145_INN  ; Z
ANDNOT V0114_INN  ; Z
ANDNOT V0143_INN  ; Z
ANDNOT V0104_INN  ; Z
OR VST80_K3_KLAPRING
ANDLD
OUT C09_0_ST_HJ3
LD TR0
AND C09_0_ST_HJ1
AND C09_0_ST_HJ2
AND C09_0_ST_HJ3
LDNOT V0146_INN
ANDNOT V0147_INN
OR VST80_K3_KLAPRING
ANDLD
OUT C09_0_ST_HJ4
; rung 24: 0-STATUS HJELP C10
LD P_On
OUT TR0
ANDNOT V0540_INN  ; Z
ANDNOT V0440_INN  ; Z
ANDNOT V0340_INN  ; Z
ANDNOT V0330_INN  ; Z
OUT C10_0_ST_HJ1
LD TR0
ANDNOT V0430_INN  ; Z
ANDNOT V0530_INN  ; Z
ANDNOT V0109_INN  ; Z
LDNOT V0342_INN  ; Z
ANDNOT V0332_INN  ; Z
OR VST80_K3_KLAPRING
ANDLD
OUT C10_0_ST_HJ2
LD TR0
LDNOT V0245_INN  ; Z
ANDNOT V0214_INN  ; Z
ANDNOT V0243_INN  ; Z
ANDNOT V0204_INN  ; Z
OR VST80_K3_KLAPRING
ANDLD
OUT C10_0_ST_HJ3
LD TR0
AND C10_0_ST_HJ1
AND C10_0_ST_HJ2
AND C10_0_ST_HJ3
LDNOT V0246_INN
ANDNOT V0247_INN
OR VST80_K3_KLAPRING
ANDLD
OUT C10_0_ST_HJ4
; rung 25: 0-STATUS HJELP C09 OG C10
LD P_On
LD C09_IND_VST80_K3  ; Z
AND C09_0_ST_HJ4
LD C10_IND_VST80_K3  ; Z
AND C10_0_ST_HJ4
ORLD
ANDLD
OUT C09_10_0_ST_HJ1

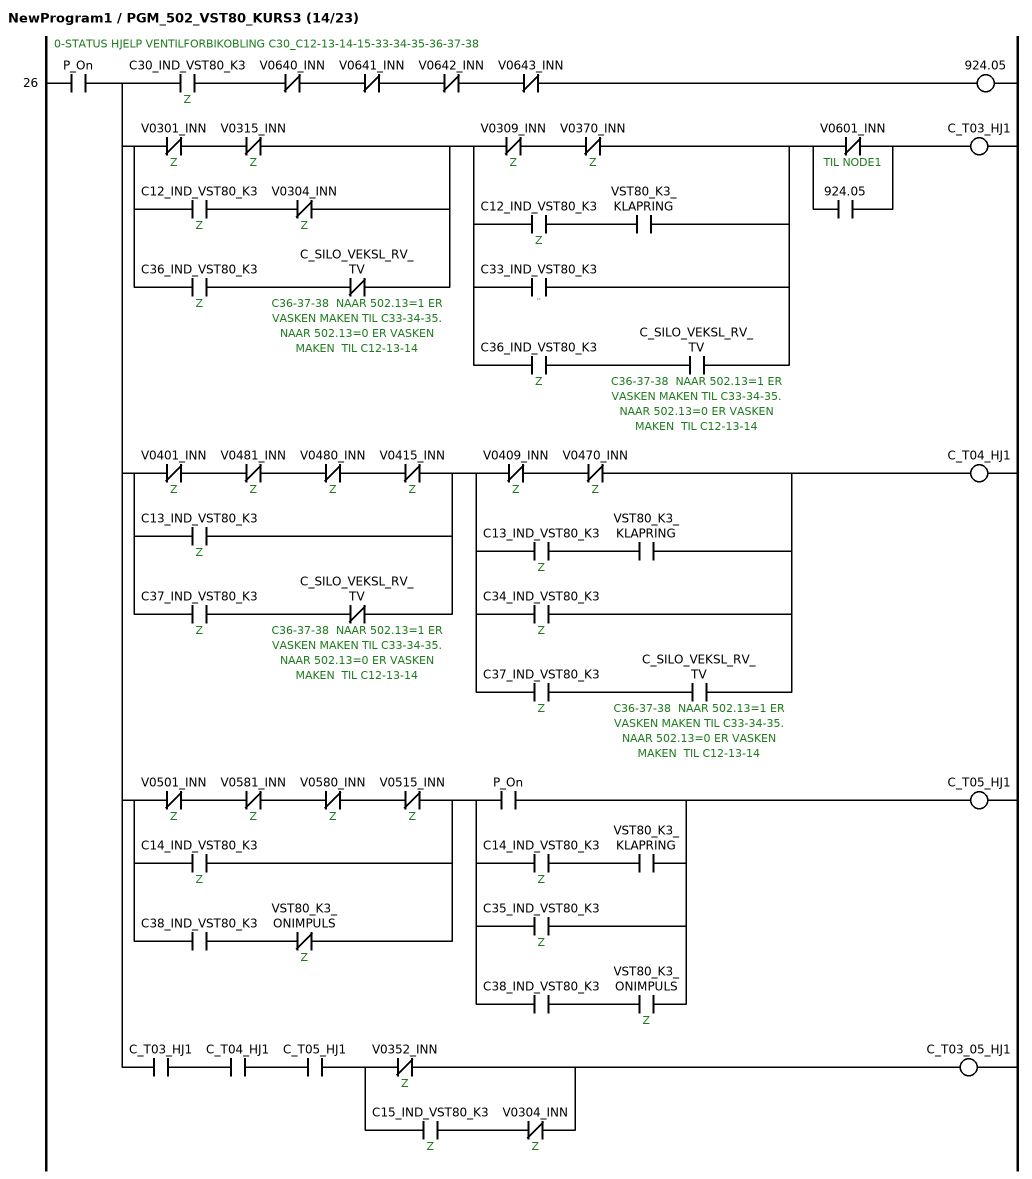
; rung 26: 0-STATUS HJELP VENTILFORBIKOBLING C30_C12-13-14-15-33-34-35-36-37-38
LD P_On
OUT TR0
AND C30_IND_VST80_K3  ; Z
ANDNOT V0640_INN
ANDNOT V0641_INN
ANDNOT V0642_INN
ANDNOT V0643_INN
OUT 924.05
LD TR0
LDNOT V0301_INN  ; Z
ANDNOT V0315_INN  ; Z
LD C12_IND_VST80_K3  ; Z
ANDNOT V0304_INN  ; Z
ORLD
LD C36_IND_VST80_K3  ; Z
ANDNOT C_SILO_VEKSL_RV_TV  ; C36-37-38  NAAR 502.13=1 ER VASKEN MAKEN TIL C33-34-35.   NAAR 502.13=0 ER VASKEN MAKEN  TIL C12-13-14
ORLD
ANDLD
LDNOT V0309_INN  ; Z
ANDNOT V0370_INN  ; Z
LD C12_IND_VST80_K3  ; Z
AND VST80_K3_KLAPRING
ORLD
OR C33_IND_VST80_K3  ; ¨
LD C36_IND_VST80_K3  ; Z
AND C_SILO_VEKSL_RV_TV  ; C36-37-38  NAAR 502.13=1 ER VASKEN MAKEN TIL C33-34-35.   NAAR 502.13=0 ER VASKEN MAKEN  TIL C12-13-14
ORLD
ANDLD
LDNOT V0601_INN  ; TIL NODE1
OR 924.05
ANDLD
OUT C_T03_HJ1
LD TR0
LDNOT V0401_INN  ; Z
ANDNOT V0481_INN  ; Z
ANDNOT V0480_INN  ; Z
ANDNOT V0415_INN  ; Z
OR C13_IND_VST80_K3  ; Z
LD C37_IND_VST80_K3  ; Z
ANDNOT C_SILO_VEKSL_RV_TV  ; C36-37-38  NAAR 502.13=1 ER VASKEN MAKEN TIL C33-34-35.   NAAR 502.13=0 ER VASKEN MAKEN  TIL C12-13-14
ORLD
ANDLD
LDNOT V0409_INN  ; Z
ANDNOT V0470_INN  ; Z
LD C13_IND_VST80_K3  ; Z
AND VST80_K3_KLAPRING
ORLD
OR C34_IND_VST80_K3  ; Z
LD C37_IND_VST80_K3  ; Z
AND C_SILO_VEKSL_RV_TV  ; C36-37-38  NAAR 502.13=1 ER VASKEN MAKEN TIL C33-34-35.   NAAR 502.13=0 ER VASKEN MAKEN  TIL C12-13-14
ORLD
ANDLD
OUT C_T04_HJ1
LD TR0
LDNOT V0501_INN  ; Z
ANDNOT V0581_INN  ; Z
ANDNOT V0580_INN  ; Z
ANDNOT V0515_INN  ; Z
OR C14_IND_VST80_K3  ; Z
LD C38_IND_VST80_K3
ANDNOT VST80_K3_ONIMPULS  ; Z
ORLD
ANDLD
LD P_On
LD C14_IND_VST80_K3  ; Z
AND VST80_K3_KLAPRING
ORLD
OR C35_IND_VST80_K3  ; Z
LD C38_IND_VST80_K3
AND VST80_K3_ONIMPULS  ; Z
ORLD
ANDLD
OUT C_T05_HJ1
LD TR0
AND C_T03_HJ1
AND C_T04_HJ1
AND C_T05_HJ1
LDNOT V0352_INN  ; Z
LD C15_IND_VST80_K3  ; Z
ANDNOT V0304_INN  ; Z
ORLD
ANDLD
OUT C_T03_05_HJ1

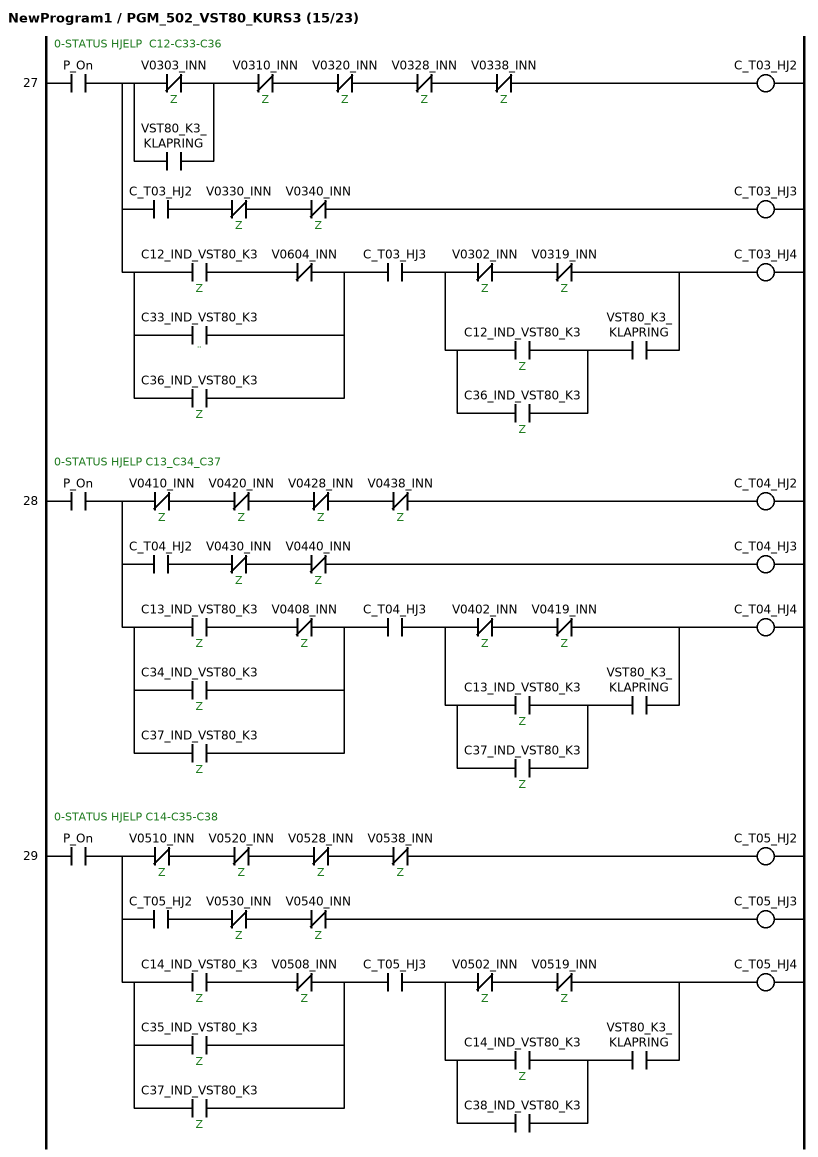
; rung 27: 0-STATUS HJELP  C12-C33-C36
LD P_On
OUT TR0
LDNOT V0303_INN  ; Z
OR VST80_K3_KLAPRING
ANDLD
ANDNOT V0310_INN  ; Z
ANDNOT V0320_INN  ; Z
ANDNOT V0328_INN  ; Z
ANDNOT V0338_INN  ; Z
OUT C_T03_HJ2
LD TR0
AND C_T03_HJ2
ANDNOT V0330_INN  ; Z
ANDNOT V0340_INN  ; Z
OUT C_T03_HJ3
LD TR0
LD C12_IND_VST80_K3  ; Z
ANDNOT V0604_INN
OR C33_IND_VST80_K3  ; ¨
OR C36_IND_VST80_K3  ; Z
ANDLD
AND C_T03_HJ3
LDNOT V0302_INN  ; Z
ANDNOT V0319_INN  ; Z
LD C12_IND_VST80_K3  ; Z
OR C36_IND_VST80_K3  ; Z
AND VST80_K3_KLAPRING
ORLD
ANDLD
OUT C_T03_HJ4
; rung 28: 0-STATUS HJELP C13_C34_C37
LD P_On
OUT TR0
ANDNOT V0410_INN  ; Z
ANDNOT V0420_INN  ; Z
ANDNOT V0428_INN  ; Z
ANDNOT V0438_INN  ; Z
OUT C_T04_HJ2
LD TR0
AND C_T04_HJ2
ANDNOT V0430_INN  ; Z
ANDNOT V0440_INN  ; Z
OUT C_T04_HJ3
LD TR0
LD C13_IND_VST80_K3  ; Z
ANDNOT V0408_INN  ; Z
OR C34_IND_VST80_K3  ; Z
OR C37_IND_VST80_K3  ; Z
ANDLD
AND C_T04_HJ3
LDNOT V0402_INN  ; Z
ANDNOT V0419_INN  ; Z
LD C13_IND_VST80_K3  ; Z
OR C37_IND_VST80_K3  ; Z
AND VST80_K3_KLAPRING
ORLD
ANDLD
OUT C_T04_HJ4
; rung 29: 0-STATUS HJELP C14-C35-C38
LD P_On
OUT TR0
ANDNOT V0510_INN  ; Z
ANDNOT V0520_INN  ; Z
ANDNOT V0528_INN  ; Z
ANDNOT V0538_INN  ; Z
OUT C_T05_HJ2
LD TR0
AND C_T05_HJ2
ANDNOT V0530_INN  ; Z
ANDNOT V0540_INN  ; Z
OUT C_T05_HJ3
LD TR0
LD C14_IND_VST80_K3  ; Z
ANDNOT V0508_INN  ; Z
OR C35_IND_VST80_K3  ; Z
OR C37_IND_VST80_K3  ; Z
ANDLD
AND C_T05_HJ3
LDNOT V0502_INN  ; Z
ANDNOT V0519_INN  ; Z
LD C14_IND_VST80_K3  ; Z
OR C38_IND_VST80_K3
AND VST80_K3_KLAPRING
ORLD
ANDLD
OUT C_T05_HJ4

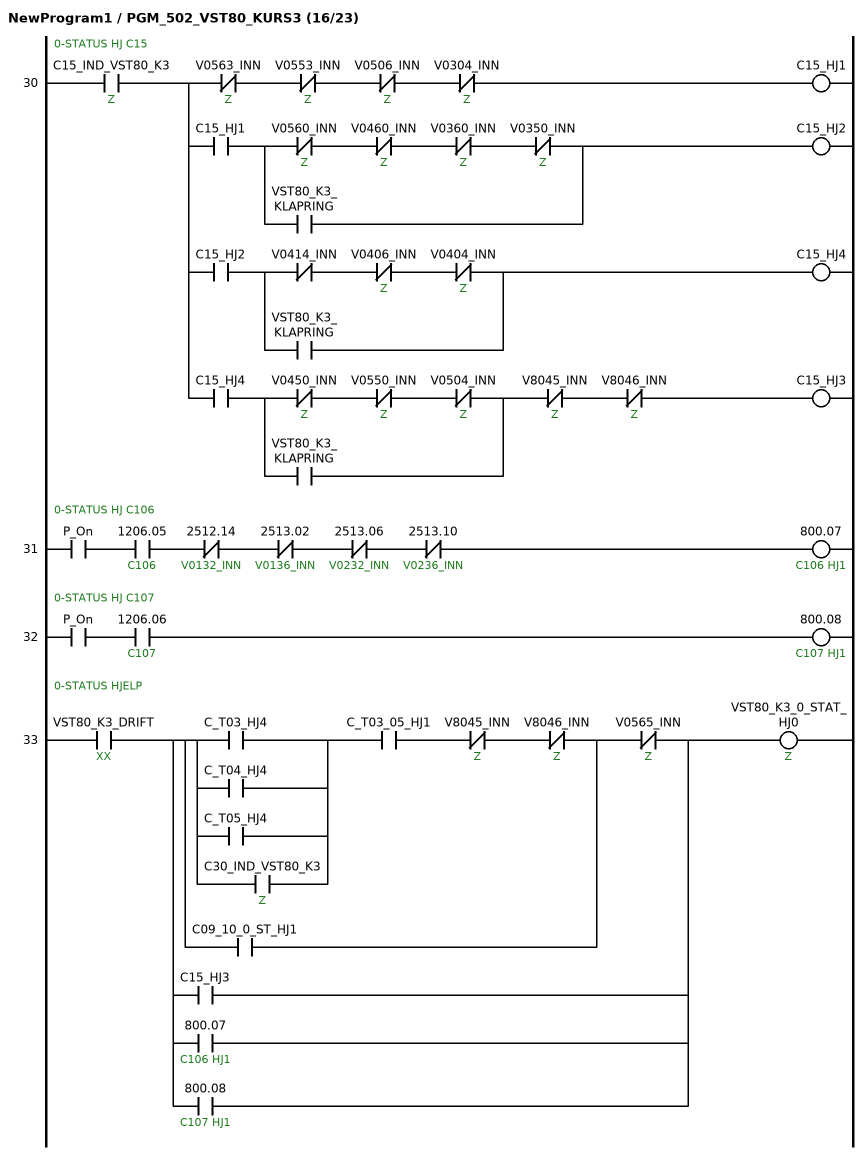
; rung 30: 0-STATUS HJ C15
LD C15_IND_VST80_K3  ; Z
OUT TR0
ANDNOT V0563_INN  ; Z
ANDNOT V0553_INN  ; Z
ANDNOT V0506_INN  ; Z
ANDNOT V0304_INN  ; Z
OUT C15_HJ1
LD TR0
AND C15_HJ1
LDNOT V0560_INN  ; Z
ANDNOT V0460_INN  ; Z
ANDNOT V0360_INN  ; Z
ANDNOT V0350_INN  ; Z
OR VST80_K3_KLAPRING
ANDLD
OUT C15_HJ2
LD TR0
AND C15_HJ2
LDNOT V0414_INN
ANDNOT V0406_INN  ; Z
ANDNOT V0404_INN  ; Z
OR VST80_K3_KLAPRING
ANDLD
OUT C15_HJ4
LD TR0
AND C15_HJ4
LDNOT V0450_INN  ; Z
ANDNOT V0550_INN  ; Z
ANDNOT V0504_INN  ; Z
OR VST80_K3_KLAPRING
ANDLD
ANDNOT V8045_INN  ; Z
ANDNOT V8046_INN  ; Z
OUT C15_HJ3
; rung 31: 0-STATUS HJ C106
LD P_On
AND 1206.05  ; C106
ANDNOT 2512.14  ; V0132_INN
ANDNOT 2513.02  ; V0136_INN
ANDNOT 2513.06  ; V0232_INN
ANDNOT 2513.10  ; V0236_INN
OUT 800.07  ; C106 HJ1
; rung 32: 0-STATUS HJ C107
LD P_On
AND 1206.06  ; C107
OUT 800.08  ; C107 HJ1
; rung 33: 0-STATUS HJELP
LD VST80_K3_DRIFT  ; XX
LD C_T03_HJ4
OR C_T04_HJ4
OR C_T05_HJ4
OR C30_IND_VST80_K3  ; Z
AND C_T03_05_HJ1
ANDNOT V8045_INN  ; Z
ANDNOT V8046_INN  ; Z
OR C09_10_0_ST_HJ1
ANDNOT V0565_INN  ; Z
OR C15_HJ3
OR 800.07  ; C106 HJ1
OR 800.08  ; C107 HJ1
ANDLD
OUT VST80_K3_0_STAT_HJ0  ; Z

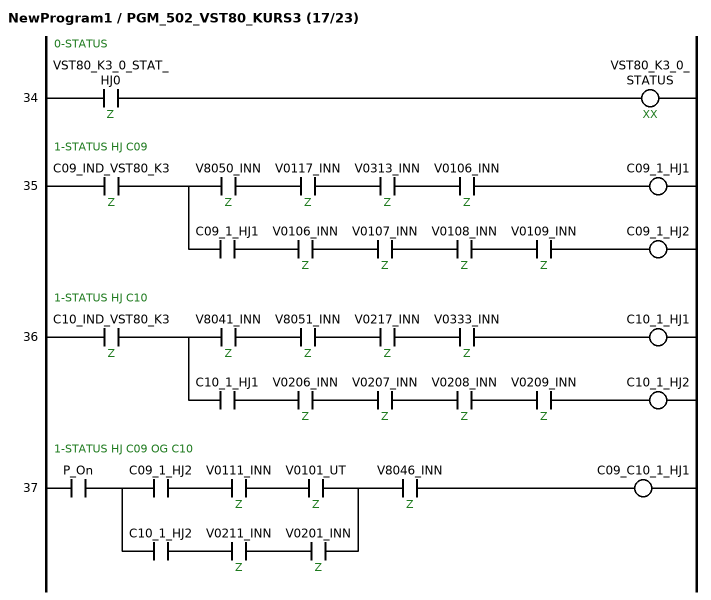
; rung 34: 0-STATUS
LD VST80_K3_0_STAT_HJ0  ; Z
OUT VST80_K3_0_STATUS  ; XX
; rung 35: 1-STATUS HJ C09
LD C09_IND_VST80_K3  ; Z
OUT TR0
AND V8050_INN  ; Z
AND V0117_INN  ; Z
AND V0313_INN  ; Z
AND V0106_INN  ; Z
OUT C09_1_HJ1
LD TR0
AND C09_1_HJ1
AND V0106_INN  ; Z
AND V0107_INN  ; Z
AND V0108_INN  ; Z
AND V0109_INN  ; Z
OUT C09_1_HJ2
; rung 36: 1-STATUS HJ C10
LD C10_IND_VST80_K3  ; Z
OUT TR0
AND V8041_INN  ; Z
AND V8051_INN  ; Z
AND V0217_INN  ; Z
AND V0333_INN  ; Z
OUT C10_1_HJ1
LD TR0
AND C10_1_HJ1
AND V0206_INN  ; Z
AND V0207_INN  ; Z
AND V0208_INN  ; Z
AND V0209_INN  ; Z
OUT C10_1_HJ2
; rung 37: 1-STATUS HJ C09 OG C10
LD P_On
LD C09_1_HJ2
AND V0111_INN  ; Z
AND V0101_UT  ; Z
LD C10_1_HJ2
AND V0211_INN  ; Z
AND V0201_INN  ; Z
ORLD
ANDLD
AND V8046_INN  ; Z
OUT C09_C10_1_HJ1

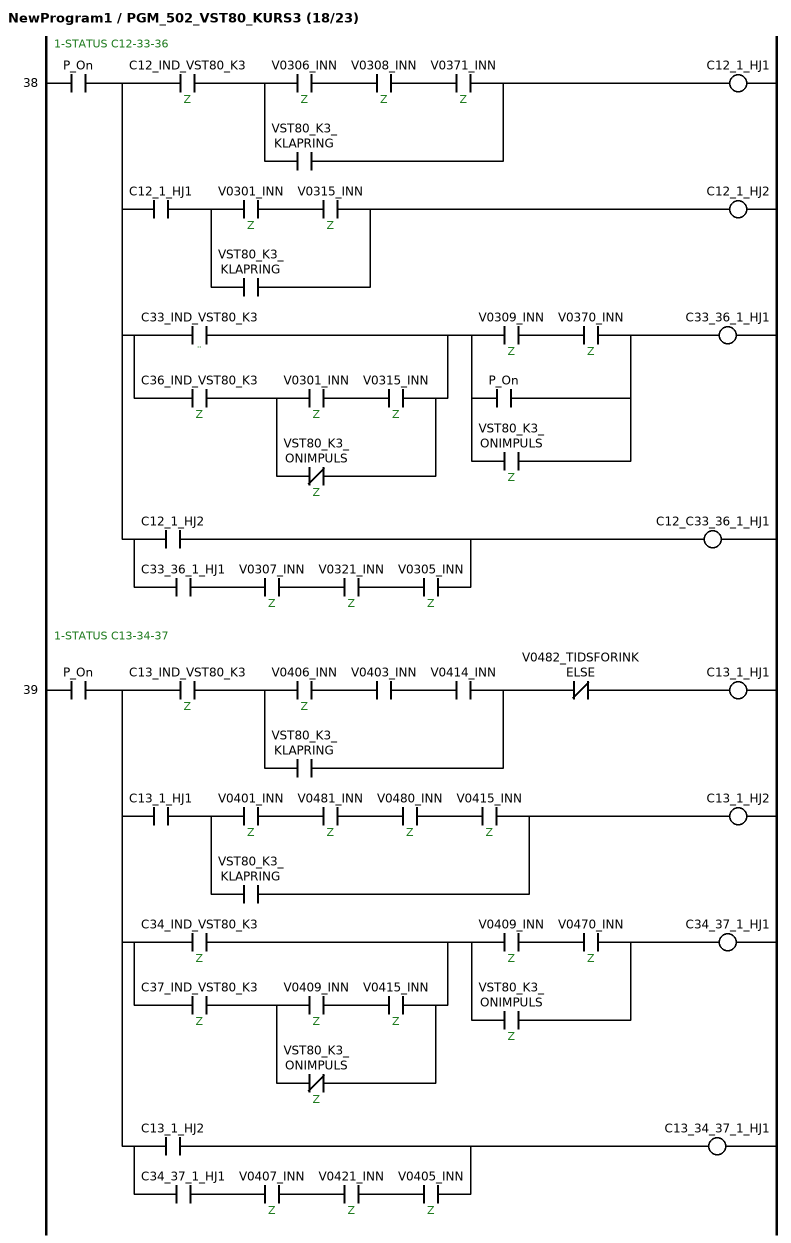
; rung 38: 1-STATUS C12-33-36
LD P_On
OUT TR0
AND C12_IND_VST80_K3  ; Z
LD V0306_INN  ; Z
AND V0308_INN  ; Z
AND V0371_INN  ; Z
OR VST80_K3_KLAPRING
ANDLD
OUT C12_1_HJ1
LD TR0
AND C12_1_HJ1
LD V0301_INN  ; Z
AND V0315_INN  ; Z
OR VST80_K3_KLAPRING
ANDLD
OUT C12_1_HJ2
LD TR0
LD C33_IND_VST80_K3  ; ¨
LD C36_IND_VST80_K3  ; Z
LD V0301_INN  ; Z
AND V0315_INN  ; Z
ORNOT VST80_K3_ONIMPULS  ; Z
ANDLD
ORLD
ANDLD
LD V0309_INN  ; Z
AND V0370_INN  ; Z
OR P_On
OR VST80_K3_ONIMPULS  ; Z
ANDLD
OUT C33_36_1_HJ1
LD TR0
LD C12_1_HJ2
LD C33_36_1_HJ1
AND V0307_INN  ; Z
AND V0321_INN  ; Z
AND V0305_INN  ; Z
ORLD
ANDLD
OUT C12_C33_36_1_HJ1
; rung 39: 1-STATUS C13-34-37
LD P_On
OUT TR0
AND C13_IND_VST80_K3  ; Z
LD V0406_INN  ; Z
AND V0403_INN
AND V0414_INN
OR VST80_K3_KLAPRING
ANDLD
ANDNOT V0482_TIDSFORINKELSE
OUT C13_1_HJ1
LD TR0
AND C13_1_HJ1
LD V0401_INN  ; Z
AND V0481_INN  ; Z
AND V0480_INN  ; Z
AND V0415_INN  ; Z
OR VST80_K3_KLAPRING
ANDLD
OUT C13_1_HJ2
LD TR0
LD C34_IND_VST80_K3  ; Z
LD C37_IND_VST80_K3  ; Z
LD V0409_INN  ; Z
AND V0415_INN  ; Z
ORNOT VST80_K3_ONIMPULS  ; Z
ANDLD
ORLD
ANDLD
LD V0409_INN  ; Z
AND V0470_INN  ; Z
OR VST80_K3_ONIMPULS  ; Z
ANDLD
OUT C34_37_1_HJ1
LD TR0
LD C13_1_HJ2
LD C34_37_1_HJ1
AND V0407_INN  ; Z
AND V0421_INN  ; Z
AND V0405_INN  ; Z
ORLD
ANDLD
OUT C13_34_37_1_HJ1

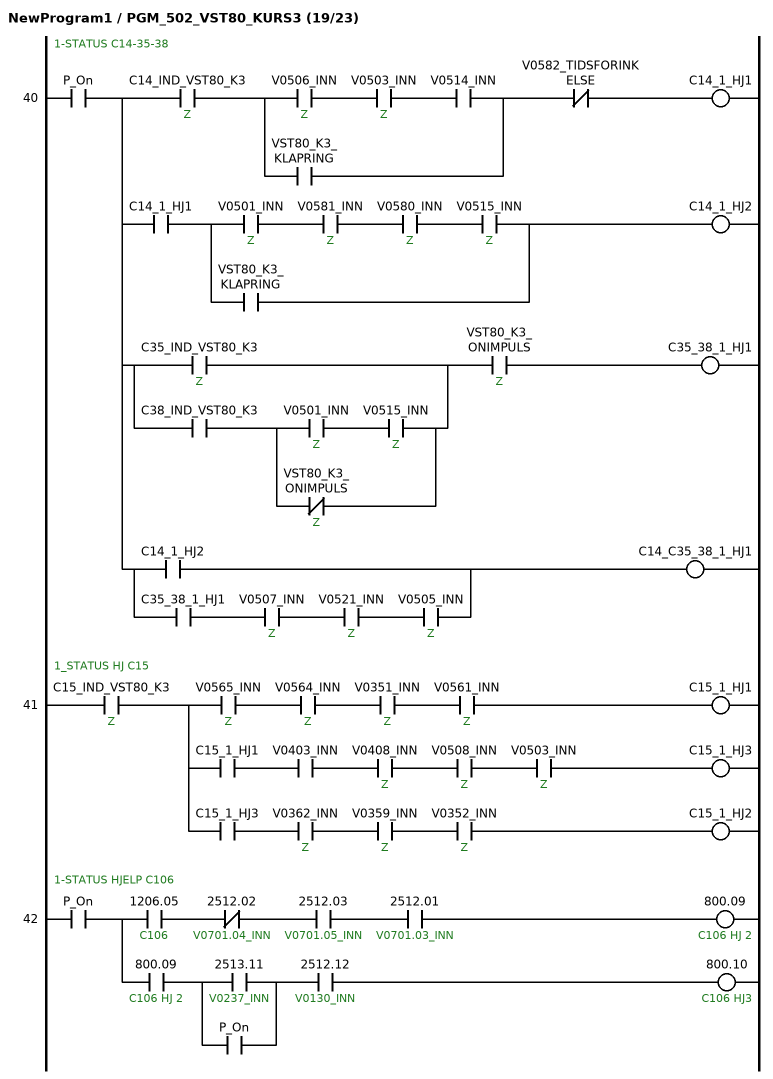
; rung 40: 1-STATUS C14-35-38
LD P_On
OUT TR0
AND C14_IND_VST80_K3  ; Z
LD V0506_INN  ; Z
AND V0503_INN  ; Z
AND V0514_INN
OR VST80_K3_KLAPRING
ANDLD
ANDNOT V0582_TIDSFORINKELSE
OUT C14_1_HJ1
LD TR0
AND C14_1_HJ1
LD V0501_INN  ; Z
AND V0581_INN  ; Z
AND V0580_INN  ; Z
AND V0515_INN  ; Z
OR VST80_K3_KLAPRING
ANDLD
OUT C14_1_HJ2
LD TR0
LD C35_IND_VST80_K3  ; Z
LD C38_IND_VST80_K3
LD V0501_INN  ; Z
AND V0515_INN  ; Z
ORNOT VST80_K3_ONIMPULS  ; Z
ANDLD
ORLD
ANDLD
AND VST80_K3_ONIMPULS  ; Z
OUT C35_38_1_HJ1
LD TR0
LD C14_1_HJ2
LD C35_38_1_HJ1
AND V0507_INN  ; Z
AND V0521_INN  ; Z
AND V0505_INN  ; Z
ORLD
ANDLD
OUT C14_C35_38_1_HJ1
; rung 41: 1_STATUS HJ C15
LD C15_IND_VST80_K3  ; Z
OUT TR0
AND V0565_INN  ; Z
AND V0564_INN  ; Z
AND V0351_INN  ; Z
AND V0561_INN  ; Z
OUT C15_1_HJ1
LD TR0
AND C15_1_HJ1
AND V0403_INN
AND V0408_INN  ; Z
AND V0508_INN  ; Z
AND V0503_INN  ; Z
OUT C15_1_HJ3
LD TR0
AND C15_1_HJ3
AND V0362_INN  ; Z
AND V0359_INN  ; Z
AND V0352_INN  ; Z
OUT C15_1_HJ2
; rung 42: 1-STATUS HJELP C106
LD P_On
OUT TR0
AND 1206.05  ; C106
ANDNOT 2512.02  ; V0701.04_INN
AND 2512.03  ; V0701.05_INN
AND 2512.01  ; V0701.03_INN
OUT 800.09  ; C106 HJ 2
LD TR0
AND 800.09  ; C106 HJ 2
LD 2513.11  ; V0237_INN
OR P_On
ANDLD
AND 2512.12  ; V0130_INN
OUT 800.10  ; C106 HJ3

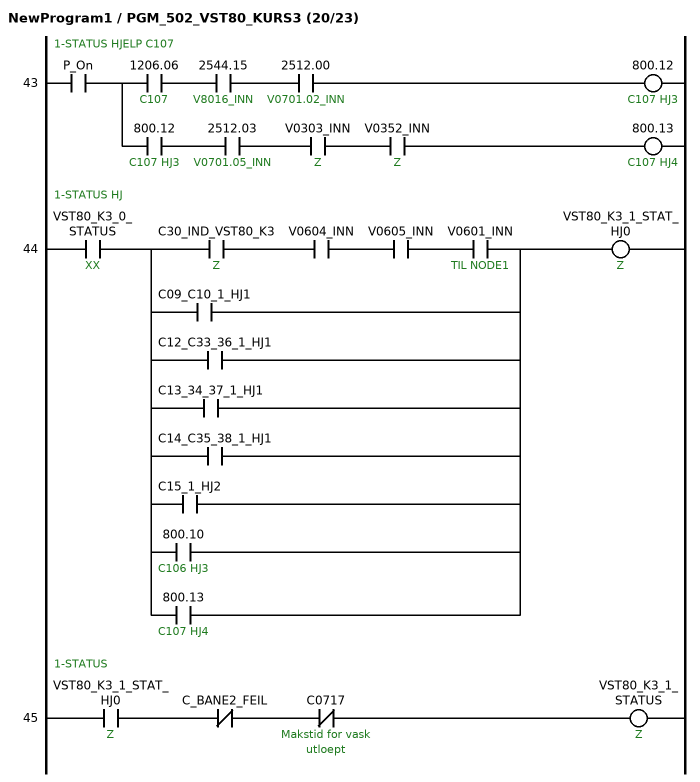
; rung 43: 1-STATUS HJELP C107
LD P_On
OUT TR0
AND 1206.06  ; C107
AND 2544.15  ; V8016_INN
AND 2512.00  ; V0701.02_INN
OUT 800.12  ; C107 HJ3
LD TR0
AND 800.12  ; C107 HJ3
AND 2512.03  ; V0701.05_INN
AND V0303_INN  ; Z
AND V0352_INN  ; Z
OUT 800.13  ; C107 HJ4
; rung 44: 1-STATUS HJ
LD VST80_K3_0_STATUS  ; XX
LD C30_IND_VST80_K3  ; Z
AND V0604_INN
AND V0605_INN
AND V0601_INN  ; TIL NODE1
OR C09_C10_1_HJ1
OR C12_C33_36_1_HJ1
OR C13_34_37_1_HJ1
OR C14_C35_38_1_HJ1
OR C15_1_HJ2
OR 800.10  ; C106 HJ3
OR 800.13  ; C107 HJ4
ANDLD
OUT VST80_K3_1_STAT_HJ0  ; Z
; rung 45: 1-STATUS
LD VST80_K3_1_STAT_HJ0  ; Z
ANDNOT C_BANE2_FEIL
ANDNOT C0717  ; Makstid for vask utloept
OUT VST80_K3_1_STATUS  ; Z

